Yaskawa INFORM job: DEMO_ROOF_SIDE_0625_3PAINT_23.JBI

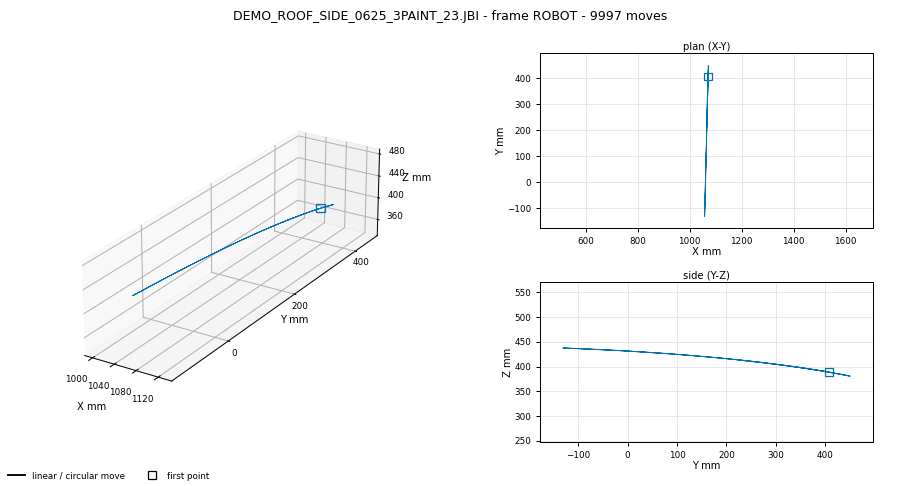
[picture p0: tool path of DEMO_ROOF_SIDE_0625_3PAINT_23.JBI in frame ROBOT, 9997 of 9997 moves have a stored position in this frame; points joined in program order, loops and branches not executed]
/JOB
//NAME DEMO_ROOF_SIDE_0625_3PAINT23
//POS
///NPOS 9997,0,0,0,0,0
///TOOL 0
///USER 0
///POSTYPE ROBOT
///RECTAN
///RCONF 1,0,0,0,0,0,0,0,0,0,0,0,0,0,0,0,0,0,0,0,0,0,0,0
C00000=1071.321,407.513,389.475,175.844,34.112,156.275
C00001=1071.313,407.267,389.517,175.839,34.102,156.273
C00002=1071.307,407.021,389.559,175.833,34.094,156.271
C00003=1071.298,406.775,389.602,175.828,34.084,156.268
C00004=1071.291,406.528,389.645,175.822,34.075,156.266
C00005=1071.284,406.282,389.687,175.818,34.066,156.264
C00006=1071.277,406.036,389.729,175.812,34.057,156.262
C00007=1071.269,405.789,389.771,175.807,34.048,156.260
C00008=1071.262,405.543,389.813,175.801,34.039,156.258
C00009=1071.254,405.297,389.855,175.796,34.030,156.256
C00010=1071.248,405.050,389.898,175.791,34.021,156.254
C00011=1071.240,404.804,389.940,175.785,34.012,156.252
C00012=1071.233,404.558,389.982,175.780,34.003,156.250
C00013=1071.225,404.311,390.025,175.775,33.995,156.248
C00014=1071.218,404.065,390.066,175.770,33.986,156.246
C00015=1071.211,403.818,390.108,175.765,33.977,156.244
C00016=1071.203,403.573,390.150,175.759,33.968,156.242
C00017=1071.196,403.326,390.192,175.754,33.959,156.240
C00018=1071.189,403.080,390.234,175.749,33.951,156.238
C00019=1071.182,402.833,390.275,175.744,33.942,156.236
C00020=1071.174,402.587,390.317,175.739,33.933,156.234
C00021=1071.166,402.341,390.359,175.733,33.925,156.232
C00022=1071.159,402.094,390.401,175.728,33.916,156.230
C00023=1071.152,401.847,390.443,175.723,33.907,156.228
C00024=1071.144,401.601,390.485,175.718,33.899,156.226
C00025=1071.137,401.354,390.526,175.713,33.890,156.224
C00026=1071.130,401.108,390.568,175.707,33.882,156.222
C00027=1071.122,400.862,390.609,175.703,33.873,156.220
C00028=1071.115,400.615,390.650,175.698,33.865,156.219
C00029=1071.109,400.370,390.692,175.692,33.856,156.217
C00030=1071.101,400.123,390.734,175.687,33.848,156.215
C00031=1071.094,399.856,390.778,175.682,33.838,156.213
C00032=1071.086,399.589,390.823,175.676,33.829,156.211
C00033=1071.078,399.323,390.868,175.671,33.820,156.208
C00034=1071.070,399.056,390.913,175.665,33.811,156.206
C00035=1071.063,398.809,390.954,175.660,33.803,156.205
C00036=1071.055,398.563,390.996,175.656,33.794,156.203
C00037=1071.049,398.316,391.038,175.650,33.786,156.201
C00038=1071.041,398.070,391.079,175.645,33.778,156.199
C00039=1071.033,397.823,391.119,175.641,33.770,156.197
C00040=1071.027,397.578,391.160,175.636,33.761,156.195
C00041=1071.019,397.331,391.201,175.630,33.753,156.193
C00042=1071.012,397.084,391.243,175.626,33.745,156.192
C00043=1071.005,396.838,391.284,175.621,33.737,156.190
C00044=1070.998,396.591,391.324,175.616,33.729,156.188
C00045=1070.991,396.345,391.365,175.611,33.720,156.186
C00046=1070.984,396.098,391.407,175.606,33.712,156.184
C00047=1070.976,395.851,391.448,175.601,33.704,156.183
C00048=1070.970,395.606,391.489,175.596,33.696,156.181
C00049=1070.962,395.359,391.530,175.591,33.688,156.179
C00050=1070.955,395.112,391.570,175.587,33.680,156.177
C00051=1070.948,394.866,391.611,175.581,33.672,156.175
C00052=1070.941,394.620,391.652,175.577,33.664,156.174
C00053=1070.934,394.372,391.692,175.572,33.656,156.172
C00054=1070.927,394.127,391.733,175.568,33.648,156.170
C00055=1070.920,393.880,391.774,175.562,33.640,156.168
C00056=1070.912,393.633,391.814,175.557,33.632,156.167
C00057=1070.905,393.387,391.855,175.553,33.624,156.165
C00058=1070.898,393.140,391.896,175.548,33.617,156.163
C00059=1070.892,392.894,391.937,175.543,33.608,156.161
C00060=1070.884,392.647,391.977,175.538,33.600,156.160
C00061=1070.877,392.401,392.018,175.534,33.593,156.158
C00062=1070.870,392.154,392.058,175.529,33.585,156.156
C00063=1070.862,391.908,392.099,175.524,33.578,156.154
C00064=1070.856,391.661,392.139,175.519,33.570,156.153
C00065=1070.849,391.414,392.179,175.515,33.562,156.151
C00066=1070.841,391.168,392.219,175.510,33.554,156.149
C00067=1070.835,390.922,392.260,175.506,33.546,156.148
C00068=1070.828,390.675,392.300,175.500,33.539,156.146
C00069=1070.820,390.428,392.340,175.496,33.531,156.144
C00070=1070.814,390.182,392.381,175.491,33.523,156.143
C00071=1070.806,389.935,392.421,175.487,33.516,156.141
C00072=1070.799,389.689,392.460,175.481,33.508,156.139
C00073=1070.793,389.442,392.501,175.477,33.501,156.138
C00074=1070.785,389.195,392.540,175.472,33.493,156.136
C00075=1070.778,388.949,392.581,175.468,33.486,156.134
C00076=1070.771,388.702,392.621,175.463,33.478,156.133
C00077=1070.764,388.455,392.661,175.459,33.471,156.131
C00078=1070.757,388.209,392.701,175.453,33.463,156.129
C00079=1070.749,387.962,392.740,175.449,33.456,156.128
C00080=1070.743,387.716,392.780,175.444,33.448,156.126
C00081=1070.735,387.469,392.820,175.440,33.441,156.124
C00082=1070.729,387.222,392.860,175.435,33.433,156.123
C00083=1070.722,386.976,392.900,175.430,33.426,156.121
C00084=1070.714,386.729,392.940,175.426,33.419,156.120
C00085=1070.708,386.483,392.980,175.421,33.411,156.118
C00086=1070.701,386.237,393.020,175.417,33.404,156.117
C00087=1070.694,385.985,393.060,175.412,33.396,156.115
C00088=1070.686,385.734,393.100,175.408,33.389,156.113
C00089=1070.680,385.483,393.141,175.402,33.382,156.112
C00090=1070.673,385.232,393.181,175.398,33.374,156.110
C00091=1070.666,384.985,393.220,175.394,33.367,156.108
C00092=1070.658,384.738,393.260,175.389,33.360,156.107
C00093=1070.652,384.492,393.300,175.385,33.352,156.105
C00094=1070.645,384.245,393.339,175.381,33.345,156.104
C00095=1070.638,383.999,393.379,175.376,33.338,156.102
C00096=1070.632,383.752,393.418,175.371,33.331,156.101
C00097=1070.625,383.505,393.458,175.366,33.323,156.099
C00098=1070.617,383.258,393.498,175.362,33.316,156.097
C00099=1070.611,383.011,393.537,175.358,33.309,156.096
C00100=1070.604,382.765,393.577,175.354,33.302,156.094
C00101=1070.597,382.518,393.615,175.349,33.295,156.093
C00102=1070.590,382.271,393.654,175.345,33.288,156.091
C00103=1070.584,382.025,393.694,175.340,33.281,156.090
C00104=1070.577,381.778,393.733,175.335,33.274,156.088
C00105=1070.570,381.532,393.773,175.331,33.266,156.087
C00106=1070.563,381.285,393.812,175.327,33.260,156.085
C00107=1070.556,381.038,393.851,175.322,33.252,156.084
C00108=1070.549,380.791,393.890,175.318,33.245,156.082
C00109=1070.543,380.544,393.930,175.314,33.239,156.081
C00110=1070.536,380.297,393.969,175.310,33.232,156.079
C00111=1070.529,380.051,394.008,175.305,33.225,156.078
C00112=1070.522,379.804,394.046,175.301,33.217,156.076
C00113=1070.515,379.557,394.085,175.296,33.211,156.075
C00114=1070.509,379.310,394.124,175.291,33.204,156.073
C00115=1070.502,379.063,394.163,175.287,33.197,156.072
C00116=1070.495,378.816,394.202,175.283,33.190,156.070
C00117=1070.488,378.570,394.241,175.279,33.183,156.069
C00118=1070.480,378.324,394.280,175.274,33.176,156.068
C00119=1070.474,378.076,394.318,175.270,33.170,156.066
C00120=1070.467,377.830,394.356,175.266,33.163,156.065
C00121=1070.460,377.583,394.395,175.262,33.156,156.063
C00122=1070.453,377.336,394.434,175.258,33.149,156.062
C00123=1070.447,377.089,394.473,175.253,33.143,156.060
C00124=1070.440,376.842,394.512,175.248,33.136,156.059
C00125=1070.433,376.595,394.551,175.244,33.129,156.057
C00126=1070.426,376.349,394.590,175.240,33.122,156.056
C00127=1070.419,376.102,394.628,175.235,33.115,156.055
C00128=1070.413,375.854,394.666,175.231,33.109,156.053
C00129=1070.406,375.607,394.705,175.227,33.102,156.052
C00130=1070.400,375.361,394.744,175.223,33.096,156.050
C00131=1070.393,375.115,394.783,175.219,33.089,156.049
C00132=1070.386,374.867,394.821,175.215,33.082,156.048
C00133=1070.380,374.620,394.860,175.210,33.075,156.046
C00134=1070.372,374.374,394.898,175.206,33.069,156.045
C00135=1070.366,374.126,394.936,175.202,33.062,156.043
C00136=1070.359,373.880,394.974,175.198,33.055,156.042
C00137=1070.353,373.633,395.013,175.194,33.049,156.041
C00138=1070.346,373.386,395.051,175.190,33.042,156.039
C00139=1070.340,373.152,395.088,175.186,33.037,156.038
C00140=1070.334,372.918,395.124,175.181,33.030,156.037
C00141=1070.327,372.684,395.160,175.177,33.024,156.035
C00142=1070.320,372.449,395.196,175.173,33.018,156.034
C00143=1070.314,372.215,395.233,175.169,33.012,156.033
C00144=1070.308,371.982,395.268,175.165,33.006,156.031
C00145=1070.301,371.747,395.305,175.161,33.000,156.030
C00146=1070.294,371.513,395.341,175.157,32.993,156.029
C00147=1070.288,371.267,395.379,175.153,32.987,156.027
C00148=1070.282,371.019,395.417,175.149,32.981,156.026
C00149=1070.274,370.773,395.455,175.145,32.974,156.025
C00150=1070.268,370.525,395.493,175.141,32.968,156.024
C00151=1070.261,370.279,395.530,175.137,32.962,156.022
C00152=1070.254,370.031,395.568,175.133,32.955,156.021
C00153=1070.248,369.785,395.607,175.129,32.949,156.019
C00154=1070.240,369.537,395.645,175.125,32.942,156.018
C00155=1070.235,369.291,395.682,175.120,32.936,156.017
C00156=1070.227,369.043,395.720,175.116,32.930,156.016
C00157=1070.221,368.796,395.758,175.112,32.924,156.014
C00158=1070.214,368.550,395.795,175.108,32.917,156.013
C00159=1070.208,368.302,395.833,175.104,32.911,156.012
C00160=1070.201,368.055,395.872,175.100,32.905,156.010
C00161=1070.194,367.809,395.909,175.096,32.898,156.009
C00162=1070.188,367.561,395.947,175.092,32.892,156.008
C00163=1070.181,367.315,395.985,175.088,32.886,156.006
C00164=1070.175,367.068,396.023,175.084,32.880,156.005
C00165=1070.168,366.821,396.059,175.080,32.874,156.004
C00166=1070.162,366.573,396.097,175.076,32.867,156.003
C00167=1070.154,366.326,396.135,175.072,32.861,156.001
C00168=1070.149,366.079,396.173,175.068,32.855,156.000
C00169=1070.141,365.832,396.210,175.064,32.849,155.999
C00170=1070.135,365.585,396.248,175.060,32.842,155.997
C00171=1070.128,365.338,396.285,175.056,32.837,155.996
C00172=1070.122,365.091,396.323,175.052,32.830,155.995
C00173=1070.115,364.844,396.360,175.048,32.824,155.994
C00174=1070.109,364.597,396.398,175.044,32.818,155.992
C00175=1070.102,364.350,396.435,175.040,32.812,155.991
C00176=1070.096,364.103,396.472,175.036,32.806,155.990
C00177=1070.089,363.855,396.510,175.032,32.800,155.989
C00178=1070.083,363.609,396.547,175.028,32.794,155.987
C00179=1070.076,363.361,396.584,175.024,32.788,155.986
C00180=1070.069,363.115,396.621,175.020,32.782,155.985
C00181=1070.063,362.867,396.659,175.016,32.776,155.984
C00182=1070.056,362.620,396.695,175.012,32.770,155.982
C00183=1070.049,362.373,396.733,175.008,32.764,155.981
C00184=1070.043,362.126,396.769,175.004,32.758,155.980
C00185=1070.036,361.879,396.808,175.000,32.752,155.979
C00186=1070.030,361.632,396.844,174.996,32.746,155.978
C00187=1070.023,361.384,396.882,174.992,32.740,155.976
C00188=1070.016,361.137,396.918,174.988,32.734,155.975
C00189=1070.010,360.890,396.954,174.984,32.728,155.974
C00190=1070.003,360.643,396.993,174.980,32.722,155.973
C00191=1069.997,360.396,397.029,174.976,32.716,155.971
C00192=1069.990,360.149,397.067,174.972,32.710,155.970
C00193=1069.983,359.902,397.103,174.969,32.705,155.969
C00194=1069.977,359.655,397.139,174.965,32.699,155.968
C00195=1069.971,359.429,397.174,174.961,32.694,155.967
C00196=1069.965,359.203,397.207,174.958,32.688,155.966
C00197=1069.960,358.978,397.240,174.955,32.683,155.965
C00198=1069.953,358.753,397.274,174.951,32.677,155.963
C00199=1069.947,358.527,397.308,174.948,32.672,155.962
C00200=1069.941,358.301,397.341,174.944,32.667,155.961
C00201=1069.936,358.075,397.375,174.941,32.661,155.960
C00202=1069.929,357.850,397.408,174.937,32.656,155.959
C00203=1069.922,357.603,397.445,174.933,32.651,155.958
C00204=1069.916,357.356,397.481,174.929,32.645,155.957
C00205=1069.909,357.108,397.518,174.925,32.639,155.956
C00206=1069.903,356.861,397.555,174.922,32.633,155.955
C00207=1069.896,356.614,397.591,174.918,32.628,155.953
C00208=1069.890,356.367,397.627,174.914,32.622,155.952
C00209=1069.883,356.119,397.664,174.910,32.616,155.951
C00210=1069.877,355.872,397.701,174.906,32.610,155.950
C00211=1069.871,355.625,397.737,174.902,32.605,155.949
C00212=1069.864,355.378,397.774,174.898,32.599,155.948
C00213=1069.857,355.130,397.810,174.895,32.594,155.946
C00214=1069.851,354.883,397.847,174.891,32.588,155.945
C00215=1069.845,354.636,397.883,174.887,32.582,155.944
C00216=1069.839,354.389,397.919,174.883,32.576,155.943
C00217=1069.832,354.141,397.955,174.880,32.571,155.942
C00218=1069.825,353.894,397.992,174.876,32.565,155.941
C00219=1069.819,353.647,398.029,174.873,32.560,155.940
C00220=1069.813,353.400,398.065,174.869,32.554,155.939
C00221=1069.806,353.152,398.100,174.865,32.548,155.937
C00222=1069.799,352.905,398.137,174.861,32.543,155.936
C00223=1069.793,352.658,398.173,174.857,32.537,155.935
C00224=1069.786,352.410,398.210,174.853,32.532,155.934
C00225=1069.780,352.163,398.246,174.850,32.526,155.933
C00226=1069.774,351.916,398.282,174.846,32.521,155.932
C00227=1069.767,351.669,398.318,174.842,32.515,155.931
C00228=1069.761,351.421,398.354,174.838,32.509,155.930
C00229=1069.754,351.174,398.390,174.834,32.504,155.929
C00230=1069.748,350.927,398.425,174.831,32.499,155.927
C00231=1069.741,350.680,398.462,174.828,32.493,155.926
C00232=1069.735,350.431,398.498,174.824,32.488,155.925
C00233=1069.728,350.184,398.534,174.820,32.482,155.924
C00234=1069.722,349.937,398.569,174.817,32.477,155.923
C00235=1069.715,349.690,398.606,174.813,32.471,155.922
C00236=1069.709,349.442,398.642,174.809,32.466,155.921
C00237=1069.702,349.195,398.678,174.805,32.460,155.920
C00238=1069.696,348.948,398.713,174.801,32.455,155.919
C00239=1069.690,348.700,398.749,174.798,32.450,155.918
C00240=1069.683,348.453,398.785,174.794,32.444,155.916
C00241=1069.677,348.206,398.821,174.790,32.439,155.915
C00242=1069.671,347.959,398.857,174.787,32.433,155.914
C00243=1069.664,347.711,398.892,174.784,32.428,155.913
C00244=1069.658,347.464,398.928,174.780,32.423,155.912
C00245=1069.651,347.216,398.963,174.776,32.417,155.911
C00246=1069.645,346.969,398.999,174.773,32.412,155.910
C00247=1069.639,346.722,399.035,174.769,32.407,155.909
C00248=1069.632,346.474,399.070,174.765,32.401,155.908
C00249=1069.626,346.226,399.106,174.761,32.396,155.907
C00250=1069.619,345.979,399.141,174.758,32.391,155.906
C00251=1069.614,345.756,399.174,174.754,32.386,155.905
C00252=1069.607,345.532,399.206,174.751,32.381,155.904
C00253=1069.602,345.309,399.238,174.749,32.376,155.903
C00254=1069.596,345.085,399.270,174.745,32.371,155.902
C00255=1069.591,344.861,399.302,174.742,32.366,155.901
C00256=1069.585,344.638,399.334,174.739,32.362,155.900
C00257=1069.579,344.413,399.367,174.735,32.357,155.899
C00258=1069.574,344.190,399.398,174.732,32.352,155.898
C00259=1069.567,343.942,399.433,174.728,32.347,155.897
C00260=1069.561,343.695,399.469,174.725,32.341,155.896
C00261=1069.554,343.447,399.504,174.721,32.337,155.895
C00262=1069.548,343.200,399.540,174.717,32.331,155.894
C00263=1069.541,342.952,399.575,174.714,32.326,155.893
C00264=1069.535,342.706,399.610,174.711,32.320,155.892
C00265=1069.528,342.458,399.645,174.707,32.316,155.891
C00266=1069.522,342.211,399.680,174.703,32.310,155.890
C00267=1069.515,341.963,399.716,174.700,32.305,155.889
C00268=1069.509,341.715,399.750,174.696,32.300,155.888
C00269=1069.503,341.468,399.786,174.692,32.295,155.887
C00270=1069.496,341.220,399.821,174.689,32.289,155.886
C00271=1069.490,340.974,399.856,174.685,32.285,155.885
C00272=1069.484,340.726,399.891,174.683,32.279,155.884
C00273=1069.478,340.478,399.926,174.679,32.274,155.883
C00274=1069.471,340.231,399.961,174.675,32.269,155.882
C00275=1069.465,339.984,399.996,174.672,32.264,155.881
C00276=1069.459,339.736,400.031,174.668,32.259,155.880
C00277=1069.452,339.488,400.066,174.664,32.254,155.879
C00278=1069.445,339.241,400.101,174.661,32.248,155.878
C00279=1069.440,338.993,400.136,174.657,32.243,155.877
C00280=1069.433,338.746,400.171,174.655,32.238,155.876
C00281=1069.427,338.499,400.206,174.651,32.233,155.875
C00282=1069.420,338.251,400.240,174.647,32.228,155.874
C00283=1069.415,338.004,400.276,174.644,32.223,155.873
C00284=1069.408,337.756,400.310,174.640,32.218,155.872
C00285=1069.402,337.508,400.345,174.637,32.213,155.871
C00286=1069.396,337.261,400.379,174.633,32.208,155.870
C00287=1069.389,337.014,400.414,174.629,32.203,155.869
C00288=1069.382,336.766,400.449,174.627,32.198,155.868
C00289=1069.376,336.518,400.484,174.623,32.193,155.867
C00290=1069.370,336.271,400.518,174.620,32.188,155.866
C00291=1069.363,336.023,400.552,174.616,32.183,155.865
C00292=1069.357,335.776,400.588,174.612,32.178,155.864
C00293=1069.351,335.528,400.622,174.609,32.173,155.863
C00294=1069.344,335.280,400.656,174.605,32.168,155.862
C00295=1069.338,335.033,400.692,174.602,32.163,155.861
C00296=1069.332,334.785,400.726,174.599,32.158,155.860
C00297=1069.326,334.537,400.760,174.596,32.153,155.859
C00298=1069.320,334.291,400.795,174.592,32.148,155.858
C00299=1069.313,334.043,400.829,174.588,32.143,155.858
C00300=1069.307,333.795,400.864,174.585,32.138,155.857
C00301=1069.301,333.548,400.898,174.581,32.133,155.856
C00302=1069.294,333.300,400.932,174.578,32.128,155.855
C00303=1069.288,333.053,400.967,174.575,32.123,155.854
C00304=1069.282,332.805,401.002,174.572,32.118,155.853
C00305=1069.276,332.558,401.036,174.568,32.113,155.852
C00306=1069.269,332.310,401.069,174.565,32.109,155.851
C00307=1069.263,332.083,401.101,174.562,32.104,155.850
C00308=1069.257,331.858,401.133,174.558,32.099,155.849
C00309=1069.252,331.631,401.164,174.555,32.095,155.848
C00310=1069.247,331.405,401.195,174.553,32.091,155.847
C00311=1069.241,331.179,401.226,174.550,32.086,155.847
C00312=1069.235,330.953,401.257,174.546,32.082,155.846
C00313=1069.229,330.727,401.289,174.543,32.077,155.845
C00314=1069.223,330.501,401.320,174.540,32.073,155.844
C00315=1069.216,330.253,401.354,174.537,32.068,155.843
C00316=1069.210,330.006,401.388,174.533,32.063,155.842
C00317=1069.204,329.757,401.421,174.530,32.058,155.841
C00318=1069.198,329.510,401.455,174.527,32.054,155.840
C00319=1069.191,329.262,401.490,174.523,32.049,155.840
C00320=1069.185,329.015,401.523,174.520,32.045,155.839
C00321=1069.178,328.767,401.558,174.516,32.040,155.838
C00322=1069.172,328.520,401.592,174.513,32.035,155.837
C00323=1069.164,328.234,401.630,174.509,32.029,155.836
C00324=1069.157,327.949,401.669,174.506,32.024,155.835
C00325=1069.150,327.663,401.708,174.502,32.019,155.834
C00326=1069.142,327.378,401.747,174.498,32.013,155.833
C00327=1069.136,327.130,401.782,174.494,32.008,155.832
C00328=1069.129,326.882,401.814,174.491,32.003,155.831
C00329=1069.123,326.634,401.849,174.488,31.999,155.830
C00330=1069.117,326.387,401.883,174.485,31.994,155.829
C00331=1069.111,326.139,401.916,174.482,31.989,155.828
C00332=1069.104,325.891,401.950,174.478,31.985,155.827
C00333=1069.098,325.644,401.984,174.475,31.980,155.826
C00334=1069.092,325.396,402.017,174.471,31.975,155.825
C00335=1069.085,325.149,402.051,174.468,31.971,155.824
C00336=1069.079,324.901,402.084,174.465,31.966,155.824
C00337=1069.072,324.653,402.118,174.462,31.961,155.823
C00338=1069.066,324.406,402.152,174.459,31.957,155.822
C00339=1069.061,324.158,402.185,174.455,31.952,155.821
C00340=1069.054,323.910,402.219,174.452,31.947,155.820
C00341=1069.048,323.662,402.252,174.448,31.943,155.819
C00342=1069.041,323.415,402.286,174.446,31.938,155.818
C00343=1069.035,323.167,402.320,174.442,31.933,155.817
C00344=1069.029,322.920,402.353,174.439,31.929,155.817
C00345=1069.023,322.672,402.386,174.436,31.924,155.816
C00346=1069.016,322.424,402.420,174.432,31.919,155.815
C00347=1069.010,322.176,402.454,174.429,31.915,155.814
C00348=1069.004,321.929,402.486,174.426,31.910,155.813
C00349=1068.998,321.681,402.520,174.423,31.905,155.812
C00350=1068.991,321.433,402.553,174.420,31.901,155.811
C00351=1068.986,321.185,402.587,174.416,31.896,155.810
C00352=1068.979,320.938,402.620,174.413,31.891,155.809
C00353=1068.974,320.690,402.654,174.410,31.887,155.809
C00354=1068.967,320.443,402.686,174.407,31.882,155.808
C00355=1068.961,320.194,402.720,174.404,31.878,155.807
C00356=1068.955,319.947,402.754,174.400,31.873,155.806
C00357=1068.948,319.700,402.786,174.397,31.868,155.805
C00358=1068.943,319.452,402.820,174.394,31.864,155.804
C00359=1068.936,319.204,402.852,174.391,31.859,155.803
C00360=1068.931,318.957,402.886,174.388,31.855,155.803
C00361=1068.924,318.708,402.920,174.385,31.850,155.802
C00362=1068.918,318.461,402.953,174.381,31.845,155.801
C00363=1068.913,318.251,402.981,174.378,31.841,155.800
C00364=1068.907,318.041,403.009,174.376,31.838,155.799
C00365=1068.903,317.830,403.037,174.374,31.833,155.799
C00366=1068.898,317.620,403.065,174.371,31.830,155.798
C00367=1068.892,317.410,403.093,174.368,31.825,155.797
C00368=1068.888,317.199,403.121,174.365,31.822,155.796
C00369=1068.882,316.989,403.149,174.362,31.817,155.796
C00370=1068.877,316.779,403.177,174.360,31.814,155.795
C00371=1068.871,316.531,403.210,174.357,31.809,155.794
C00372=1068.865,316.283,403.243,174.354,31.805,155.793
C00373=1068.859,316.036,403.276,174.351,31.800,155.792
C00374=1068.853,315.788,403.309,174.347,31.795,155.791
C00375=1068.847,315.540,403.342,174.344,31.791,155.791
C00376=1068.841,315.293,403.375,174.341,31.786,155.790
C00377=1068.835,315.045,403.408,174.338,31.781,155.789
C00378=1068.829,314.797,403.441,174.335,31.777,155.788
C00379=1068.823,314.549,403.474,174.332,31.772,155.787
C00380=1068.817,314.302,403.507,174.329,31.768,155.786
C00381=1068.811,314.053,403.539,174.325,31.764,155.785
C00382=1068.804,313.805,403.572,174.323,31.759,155.785
C00383=1068.798,313.558,403.605,174.320,31.755,155.784
C00384=1068.791,313.310,403.638,174.316,31.750,155.783
C00385=1068.785,313.062,403.670,174.313,31.746,155.782
C00386=1068.779,312.814,403.702,174.310,31.742,155.781
C00387=1068.773,312.567,403.735,174.307,31.737,155.781
C00388=1068.766,312.319,403.767,174.304,31.733,155.780
C00389=1068.760,312.071,403.799,174.301,31.728,155.779
C00390=1068.754,311.823,403.832,174.297,31.724,155.778
C00391=1068.747,311.576,403.865,174.294,31.719,155.777
C00392=1068.741,311.328,403.897,174.291,31.715,155.776
C00393=1068.735,311.080,403.930,174.289,31.711,155.776
C00394=1068.729,310.833,403.962,174.285,31.706,155.775
C00395=1068.723,310.584,403.994,174.282,31.702,155.774
C00396=1068.716,310.337,404.027,174.279,31.697,155.773
C00397=1068.709,310.089,404.059,174.275,31.693,155.772
C00398=1068.703,309.841,404.091,174.273,31.689,155.772
C00399=1068.697,309.594,404.124,174.270,31.684,155.771
C00400=1068.691,309.345,404.156,174.267,31.680,155.770
C00401=1068.685,309.098,404.189,174.263,31.676,155.769
C00402=1068.679,308.850,404.221,174.260,31.671,155.768
C00403=1068.672,308.602,404.253,174.258,31.667,155.768
C00404=1068.666,308.354,404.285,174.255,31.663,155.767
C00405=1068.660,308.107,404.318,174.251,31.658,155.766
C00406=1068.654,307.859,404.349,174.248,31.654,155.765
C00407=1068.648,307.611,404.382,174.245,31.649,155.764
C00408=1068.642,307.363,404.414,174.243,31.645,155.764
C00409=1068.635,307.115,404.446,174.239,31.641,155.763
C00410=1068.629,306.868,404.478,174.236,31.636,155.762
C00411=1068.623,306.619,404.510,174.233,31.632,155.761
C00412=1068.617,306.372,404.543,174.230,31.628,155.760
C00413=1068.611,306.124,404.575,174.227,31.623,155.760
C00414=1068.604,305.876,404.606,174.224,31.619,155.759
C00415=1068.598,305.629,404.639,174.221,31.615,155.758
C00416=1068.592,305.381,404.671,174.218,31.610,155.757
C00417=1068.586,305.132,404.703,174.215,31.606,155.756
C00418=1068.580,304.885,404.734,174.212,31.602,155.756
C00419=1068.575,304.658,404.764,174.209,31.597,155.755
C00420=1068.569,304.430,404.793,174.206,31.594,155.754
C00421=1068.564,304.203,404.823,174.203,31.589,155.753
C00422=1068.558,303.975,404.852,174.201,31.586,155.753
C00423=1068.552,303.748,404.881,174.199,31.581,155.752
C00424=1068.547,303.521,404.910,174.196,31.578,155.751
C00425=1068.541,303.293,404.940,174.193,31.573,155.750
C00426=1068.535,303.066,404.969,174.190,31.570,155.750
C00427=1068.529,302.817,405.001,174.187,31.565,155.749
C00428=1068.523,302.569,405.033,174.184,31.561,155.748
C00429=1068.518,302.322,405.065,174.181,31.557,155.747
C00430=1068.511,302.074,405.096,174.178,31.552,155.747
C00431=1068.505,301.826,405.129,174.175,31.548,155.746
C00432=1068.499,301.579,405.160,174.173,31.544,155.745
C00433=1068.493,301.331,405.192,174.169,31.539,155.744
C00434=1068.487,301.083,405.224,174.166,31.535,155.743
C00435=1068.481,300.835,405.256,174.163,31.531,155.743
C00436=1068.475,300.587,405.288,174.160,31.526,155.742
C00437=1068.469,300.339,405.319,174.158,31.522,155.741
C00438=1068.463,300.092,405.351,174.155,31.518,155.740
C00439=1068.457,299.843,405.383,174.152,31.514,155.739
C00440=1068.451,299.596,405.414,174.148,31.509,155.739
C00441=1068.445,299.348,405.446,174.146,31.505,155.738
C00442=1068.440,299.099,405.477,174.143,31.500,155.737
C00443=1068.433,298.852,405.508,174.140,31.496,155.736
C00444=1068.427,298.604,405.540,174.137,31.492,155.735
C00445=1068.422,298.356,405.572,174.134,31.488,155.735
C00446=1068.415,298.108,405.603,174.132,31.483,155.734
C00447=1068.410,297.861,405.635,174.128,31.479,155.733
C00448=1068.404,297.612,405.667,174.125,31.474,155.732
C00449=1068.397,297.364,405.698,174.122,31.470,155.731
C00450=1068.392,297.116,405.729,174.120,31.466,155.731
C00451=1068.385,296.869,405.761,174.117,31.462,155.730
C00452=1068.380,296.621,405.792,174.114,31.457,155.729
C00453=1068.374,296.373,405.823,174.111,31.453,155.728
C00454=1068.368,296.124,405.855,174.108,31.449,155.728
C00455=1068.361,295.877,405.886,174.105,31.445,155.727
C00456=1068.355,295.629,405.917,174.102,31.440,155.726
C00457=1068.350,295.381,405.949,174.099,31.436,155.725
C00458=1068.343,295.133,405.980,174.096,31.432,155.725
C00459=1068.337,294.885,406.010,174.094,31.428,155.724
C00460=1068.331,294.637,406.042,174.091,31.424,155.723
C00461=1068.325,294.389,406.073,174.088,31.419,155.722
C00462=1068.319,294.141,406.104,174.085,31.416,155.722
C00463=1068.313,293.893,406.136,174.082,31.411,155.721
C00464=1068.307,293.645,406.167,174.079,31.407,155.720
C00465=1068.300,293.397,406.198,174.076,31.402,155.719
C00466=1068.294,293.150,406.228,174.073,31.399,155.719
C00467=1068.288,292.901,406.260,174.070,31.394,155.718
C00468=1068.282,292.654,406.291,174.068,31.390,155.717
C00469=1068.276,292.406,406.322,174.065,31.386,155.716
C00470=1068.270,292.158,406.353,174.062,31.382,155.716
C00471=1068.264,291.910,406.385,174.059,31.378,155.715
C00472=1068.258,291.662,406.415,174.057,31.373,155.714
C00473=1068.252,291.413,406.446,174.054,31.370,155.713
C00474=1068.246,291.166,406.477,174.051,31.365,155.712
C00475=1068.240,290.946,406.504,174.048,31.361,155.712
C00476=1068.235,290.726,406.532,174.045,31.358,155.711
C00477=1068.230,290.505,406.559,174.044,31.354,155.710
C00478=1068.225,290.285,406.586,174.041,31.350,155.710
C00479=1068.219,290.066,406.614,174.038,31.346,155.709
C00480=1068.214,289.846,406.641,174.035,31.343,155.708
C00481=1068.208,289.626,406.668,174.034,31.339,155.708
C00482=1068.203,289.405,406.696,174.031,31.336,155.707
C00483=1068.197,289.158,406.726,174.028,31.332,155.706
C00484=1068.191,288.910,406.758,174.025,31.327,155.706
C00485=1068.185,288.662,406.788,174.022,31.323,155.705
C00486=1068.178,288.413,406.819,174.020,31.319,155.704
C00487=1068.173,288.165,406.849,174.017,31.315,155.703
C00488=1068.166,287.917,406.880,174.014,31.311,155.703
C00489=1068.160,287.670,406.911,174.011,31.307,155.702
C00490=1068.154,287.422,406.941,174.009,31.303,155.701
C00491=1068.148,287.173,406.972,174.006,31.299,155.700
C00492=1068.142,286.926,407.002,174.003,31.294,155.700
C00493=1068.136,286.677,407.033,174.000,31.290,155.699
C00494=1068.130,286.429,407.063,173.997,31.286,155.698
C00495=1068.124,286.181,407.094,173.994,31.282,155.698
C00496=1068.117,285.933,407.124,173.991,31.278,155.697
C00497=1068.112,285.685,407.155,173.988,31.274,155.696
C00498=1068.106,285.437,407.185,173.986,31.270,155.695
C00499=1068.099,285.189,407.216,173.983,31.265,155.695
C00500=1068.094,284.941,407.246,173.980,31.262,155.694
C00501=1068.088,284.693,407.277,173.977,31.257,155.693
C00502=1068.081,284.445,407.307,173.975,31.253,155.692
C00503=1068.076,284.197,407.338,173.972,31.249,155.692
C00504=1068.069,283.949,407.367,173.969,31.245,155.691
C00505=1068.063,283.701,407.398,173.966,31.241,155.690
C00506=1068.057,283.453,407.428,173.964,31.237,155.689
C00507=1068.051,283.205,407.459,173.961,31.233,155.689
C00508=1068.045,282.957,407.490,173.958,31.228,155.688
C00509=1068.039,282.709,407.520,173.955,31.225,155.687
C00510=1068.033,282.461,407.550,173.953,31.220,155.686
C00511=1068.027,282.212,407.580,173.950,31.216,155.686
C00512=1068.021,281.964,407.611,173.948,31.212,155.685
C00513=1068.015,281.716,407.641,173.945,31.208,155.684
C00514=1068.009,281.468,407.671,173.943,31.204,155.684
C00515=1068.003,281.221,407.701,173.940,31.200,155.683
C00516=1067.997,280.972,407.731,173.937,31.196,155.682
C00517=1067.991,280.724,407.761,173.934,31.192,155.681
C00518=1067.985,280.476,407.792,173.932,31.187,155.681
C00519=1067.979,280.228,407.822,173.929,31.184,155.680
C00520=1067.974,279.980,407.852,173.926,31.180,155.679
C00521=1067.967,279.732,407.882,173.923,31.175,155.678
C00522=1067.961,279.484,407.912,173.921,31.172,155.678
C00523=1067.955,279.235,407.942,173.918,31.167,155.677
C00524=1067.949,278.988,407.972,173.915,31.163,155.676
C00525=1067.942,278.739,408.002,173.912,31.159,155.676
C00526=1067.937,278.491,408.032,173.910,31.155,155.675
C00527=1067.930,278.243,408.062,173.907,31.151,155.674
C00528=1067.925,277.995,408.091,173.904,31.147,155.673
C00529=1067.919,277.747,408.122,173.901,31.143,155.673
C00530=1067.913,277.499,408.152,173.899,31.139,155.672
C00531=1067.907,277.284,408.178,173.897,31.135,155.671
C00532=1067.902,277.069,408.203,173.894,31.132,155.671
C00533=1067.897,276.854,408.229,173.892,31.128,155.670
C00534=1067.891,276.639,408.255,173.890,31.125,155.669
C00535=1067.886,276.425,408.281,173.888,31.121,155.669
C00536=1067.881,276.209,408.307,173.885,31.118,155.668
C00537=1067.876,275.995,408.332,173.883,31.115,155.668
C00538=1067.870,275.780,408.358,173.880,31.111,155.667
C00539=1067.865,275.531,408.388,173.878,31.107,155.666
C00540=1067.859,275.284,408.418,173.875,31.103,155.666
C00541=1067.853,275.036,408.447,173.872,31.099,155.665
C00542=1067.847,274.787,408.477,173.870,31.094,155.664
C00543=1067.841,274.540,408.507,173.867,31.091,155.663
C00544=1067.835,274.291,408.537,173.865,31.086,155.663
C00545=1067.829,274.043,408.566,173.862,31.083,155.662
C00546=1067.822,273.794,408.596,173.860,31.078,155.661
C00547=1067.817,273.546,408.626,173.857,31.074,155.660
C00548=1067.811,273.298,408.655,173.854,31.071,155.660
C00549=1067.805,273.050,408.685,173.851,31.066,155.659
C00550=1067.799,272.802,408.714,173.849,31.062,155.658
C00551=1067.793,272.554,408.744,173.846,31.058,155.658
C00552=1067.787,272.305,408.773,173.843,31.054,155.657
C00553=1067.780,272.058,408.803,173.840,31.050,155.656
C00554=1067.775,271.809,408.832,173.839,31.046,155.655
C00555=1067.769,271.561,408.861,173.836,31.042,155.655
C00556=1067.763,271.313,408.891,173.833,31.038,155.654
C00557=1067.756,271.065,408.921,173.831,31.034,155.653
C00558=1067.751,270.817,408.950,173.828,31.030,155.653
C00559=1067.745,270.569,408.979,173.825,31.026,155.652
C00560=1067.738,270.321,409.009,173.822,31.022,155.651
C00561=1067.733,270.072,409.038,173.820,31.018,155.650
C00562=1067.727,269.824,409.067,173.818,31.014,155.650
C00563=1067.721,269.576,409.097,173.815,31.010,155.649
C00564=1067.715,269.327,409.126,173.812,31.006,155.648
C00565=1067.709,269.079,409.155,173.810,31.002,155.648
C00566=1067.703,268.831,409.185,173.807,30.998,155.647
C00567=1067.697,268.583,409.214,173.804,30.994,155.646
C00568=1067.691,268.335,409.243,173.802,30.990,155.646
C00569=1067.684,268.087,409.272,173.800,30.986,155.645
C00570=1067.679,267.838,409.301,173.797,30.982,155.644
C00571=1067.673,267.590,409.330,173.794,30.978,155.644
C00572=1067.666,267.342,409.359,173.792,30.974,155.643
C00573=1067.660,267.094,409.388,173.789,30.970,155.642
C00574=1067.655,266.845,409.418,173.786,30.966,155.641
C00575=1067.648,266.597,409.447,173.783,30.962,155.641
C00576=1067.642,266.349,409.476,173.782,30.958,155.640
C00577=1067.636,266.101,409.505,173.779,30.954,155.639
C00578=1067.630,265.852,409.535,173.776,30.950,155.639
C00579=1067.624,265.604,409.564,173.774,30.946,155.638
C00580=1067.618,265.356,409.593,173.771,30.942,155.637
C00581=1067.612,265.107,409.621,173.769,30.938,155.636
C00582=1067.606,264.859,409.651,173.766,30.934,155.636
C00583=1067.600,264.611,409.680,173.764,30.930,155.635
C00584=1067.594,264.363,409.709,173.761,30.926,155.634
C00585=1067.588,264.115,409.738,173.758,30.922,155.634
C00586=1067.582,263.867,409.766,173.756,30.918,155.633
C00587=1067.578,263.653,409.792,173.754,30.915,155.632
C00588=1067.572,263.440,409.817,173.752,30.911,155.632
C00589=1067.567,263.227,409.841,173.749,30.908,155.631
C00590=1067.561,263.014,409.866,173.748,30.904,155.631
C00591=1067.556,262.801,409.890,173.745,30.901,155.630
C00592=1067.551,262.588,409.915,173.743,30.898,155.629
C00593=1067.545,262.374,409.939,173.741,30.894,155.629
C00594=1067.540,262.162,409.964,173.739,30.891,155.628
C00595=1067.534,261.914,409.993,173.736,30.887,155.627
C00596=1067.528,261.665,410.021,173.733,30.883,155.627
C00597=1067.522,261.417,410.050,173.731,30.879,155.626
C00598=1067.516,261.168,410.079,173.729,30.875,155.625
C00599=1067.510,260.920,410.108,173.726,30.871,155.625
C00600=1067.504,260.671,410.136,173.723,30.867,155.624
C00601=1067.497,260.423,410.165,173.721,30.863,155.623
C00602=1067.491,260.175,410.194,173.719,30.860,155.623
C00603=1067.485,259.927,410.222,173.716,30.855,155.622
C00604=1067.479,259.679,410.251,173.713,30.851,155.621
C00605=1067.473,259.430,410.279,173.711,30.848,155.621
C00606=1067.467,259.182,410.308,173.709,30.844,155.620
C00607=1067.461,258.933,410.336,173.706,30.839,155.619
C00608=1067.455,258.685,410.365,173.704,30.836,155.618
C00609=1067.449,258.438,410.393,173.701,30.832,155.618
C00610=1067.443,258.189,410.421,173.698,30.828,155.617
C00611=1067.436,257.941,410.450,173.696,30.824,155.616
C00612=1067.430,257.692,410.478,173.694,30.820,155.616
C00613=1067.424,257.444,410.507,173.691,30.816,155.615
C00614=1067.419,257.196,410.535,173.688,30.812,155.614
C00615=1067.413,256.947,410.564,173.687,30.808,155.614
C00616=1067.406,256.699,410.592,173.684,30.804,155.613
C00617=1067.400,256.450,410.620,173.681,30.800,155.612
C00618=1067.394,256.202,410.649,173.678,30.796,155.612
C00619=1067.388,255.954,410.677,173.677,30.792,155.611
C00620=1067.382,255.706,410.706,173.674,30.788,155.610
C00621=1067.376,255.457,410.734,173.671,30.784,155.610
C00622=1067.370,255.210,410.762,173.669,30.780,155.609
C00623=1067.364,254.961,410.791,173.667,30.776,155.608
C00624=1067.358,254.712,410.819,173.664,30.772,155.607
C00625=1067.352,254.463,410.847,173.662,30.769,155.607
C00626=1067.347,254.216,410.876,173.659,30.764,155.606
C00627=1067.340,253.968,410.904,173.657,30.760,155.605
C00628=1067.334,253.719,410.932,173.654,30.757,155.605
C00629=1067.329,253.471,410.960,173.652,30.752,155.604
C00630=1067.323,253.222,410.988,173.650,30.749,155.603
C00631=1067.316,252.974,411.017,173.647,30.745,155.603
C00632=1067.310,252.726,411.045,173.645,30.740,155.602
C00633=1067.304,252.477,411.073,173.642,30.736,155.601
C00634=1067.298,252.229,411.101,173.640,30.733,155.600
C00635=1067.293,251.981,411.129,173.638,30.728,155.600
C00636=1067.286,251.732,411.157,173.635,30.724,155.599
C00637=1067.281,251.484,411.185,173.633,30.721,155.598
C00638=1067.275,251.235,411.213,173.631,30.716,155.598
C00639=1067.269,250.987,411.242,173.628,30.712,155.597
C00640=1067.263,250.739,411.269,173.625,30.709,155.596
C00641=1067.257,250.490,411.297,173.624,30.704,155.596
C00642=1067.252,250.242,411.325,173.621,30.700,155.595
C00643=1067.246,250.028,411.350,173.619,30.697,155.594
C00644=1067.241,249.814,411.373,173.616,30.693,155.594
C00645=1067.236,249.599,411.399,173.615,30.690,155.593
C00646=1067.231,249.385,411.422,173.613,30.687,155.592
C00647=1067.226,249.171,411.446,173.611,30.683,155.592
C00648=1067.221,248.956,411.471,173.608,30.680,155.591
C00649=1067.216,248.742,411.495,173.607,30.676,155.591
C00650=1067.211,248.527,411.519,173.605,30.673,155.590
C00651=1067.205,248.279,411.546,173.602,30.669,155.589
C00652=1067.199,248.031,411.574,173.600,30.665,155.589
C00653=1067.193,247.783,411.602,173.598,30.661,155.588
C00654=1067.187,247.534,411.630,173.595,30.656,155.587
C00655=1067.182,247.286,411.658,173.593,30.653,155.586
C00656=1067.175,247.038,411.686,173.591,30.649,155.586
C00657=1067.170,246.789,411.714,173.588,30.644,155.585
C00658=1067.164,246.540,411.742,173.586,30.641,155.584
C00659=1067.158,246.292,411.769,173.584,30.636,155.584
C00660=1067.152,246.044,411.797,173.581,30.632,155.583
C00661=1067.146,245.796,411.825,173.578,30.629,155.582
C00662=1067.140,245.547,411.853,173.577,30.625,155.582
C00663=1067.135,245.299,411.880,173.574,30.620,155.581
C00664=1067.129,245.050,411.908,173.571,30.616,155.580
C00665=1067.123,244.802,411.935,173.570,30.613,155.580
C00666=1067.117,244.553,411.963,173.567,30.608,155.579
C00667=1067.111,244.305,411.990,173.564,30.604,155.578
C00668=1067.104,244.057,412.018,173.563,30.601,155.577
C00669=1067.099,243.809,412.046,173.560,30.596,155.577
C00670=1067.092,243.560,412.073,173.557,30.592,155.576
C00671=1067.087,243.312,412.101,173.556,30.589,155.575
C00672=1067.081,243.062,412.128,173.553,30.584,155.575
C00673=1067.075,242.814,412.156,173.551,30.581,155.574
C00674=1067.069,242.567,412.183,173.549,30.577,155.573
C00675=1067.064,242.317,412.211,173.546,30.572,155.572
C00676=1067.058,242.070,412.238,173.544,30.569,155.572
C00677=1067.051,241.821,412.265,173.542,30.565,155.571
C00678=1067.045,241.573,412.293,173.539,30.561,155.571
C00679=1067.039,241.323,412.320,173.537,30.557,155.570
C00680=1067.033,241.076,412.348,173.535,30.553,155.569
C00681=1067.027,240.827,412.375,173.533,30.549,155.568
C00682=1067.021,240.579,412.402,173.530,30.545,155.568
C00683=1067.015,240.330,412.430,173.528,30.541,155.567
C00684=1067.009,240.082,412.457,173.526,30.537,155.566
C00685=1067.003,239.833,412.484,173.523,30.533,155.566
C00686=1066.997,239.585,412.511,173.521,30.529,155.565
C00687=1066.992,239.336,412.539,173.519,30.525,155.564
C00688=1066.985,239.088,412.566,173.516,30.521,155.564
C00689=1066.979,238.839,412.593,173.515,30.517,155.563
C00690=1066.973,238.590,412.620,173.512,30.513,155.562
C00691=1066.967,238.343,412.647,173.509,30.509,155.561
C00692=1066.962,238.094,412.675,173.508,30.505,155.561
C00693=1066.955,237.845,412.702,173.505,30.501,155.560
C00694=1066.949,237.597,412.729,173.503,30.497,155.559
C00695=1066.943,237.348,412.756,173.501,30.493,155.559
C00696=1066.937,237.100,412.783,173.498,30.489,155.558
C00697=1066.931,236.852,412.810,173.496,30.485,155.557
C00698=1066.925,236.603,412.838,173.494,30.481,155.557
C00699=1066.921,236.386,412.861,173.492,30.478,155.556
C00700=1066.915,236.168,412.884,173.490,30.474,155.555
C00701=1066.910,235.951,412.908,173.489,30.471,155.555
C00702=1066.905,235.733,412.932,173.486,30.467,155.554
C00703=1066.900,235.516,412.955,173.484,30.463,155.554
C00704=1066.894,235.298,412.979,173.482,30.460,155.553
C00705=1066.889,235.080,413.003,173.481,30.457,155.552
C00706=1066.884,234.863,413.026,173.478,30.453,155.552
C00707=1066.878,234.615,413.054,173.476,30.449,155.551
C00708=1066.872,234.366,413.081,173.474,30.445,155.550
C00709=1066.866,234.118,413.107,173.472,30.441,155.550
C00710=1066.860,233.870,413.134,173.469,30.437,155.549
C00711=1066.855,233.621,413.161,173.467,30.433,155.548
C00712=1066.848,233.372,413.188,173.465,30.429,155.548
C00713=1066.842,233.124,413.215,173.462,30.425,155.547
C00714=1066.836,232.876,413.242,173.461,30.421,155.546
C00715=1066.830,232.627,413.269,173.458,30.417,155.546
C00716=1066.824,232.379,413.295,173.456,30.413,155.545
C00717=1066.818,232.130,413.322,173.454,30.409,155.544
C00718=1066.813,231.882,413.349,173.452,30.405,155.543
C00719=1066.806,231.633,413.376,173.450,30.401,155.543
C00720=1066.800,231.384,413.402,173.448,30.397,155.542
C00721=1066.795,231.136,413.429,173.445,30.393,155.541
C00722=1066.789,230.888,413.456,173.443,30.389,155.541
C00723=1066.783,230.639,413.483,173.441,30.385,155.540
C00724=1066.777,230.390,413.509,173.438,30.381,155.539
C00725=1066.771,230.142,413.536,173.437,30.377,155.538
C00726=1066.765,229.894,413.563,173.434,30.373,155.538
C00727=1066.759,229.645,413.589,173.432,30.369,155.537
C00728=1066.753,229.396,413.616,173.430,30.365,155.536
C00729=1066.748,229.147,413.642,173.428,30.361,155.536
C00730=1066.742,228.899,413.669,173.425,30.357,155.535
C00731=1066.735,228.650,413.695,173.424,30.353,155.534
C00732=1066.729,228.402,413.722,173.421,30.349,155.534
C00733=1066.723,228.153,413.749,173.419,30.345,155.533
C00734=1066.717,227.905,413.775,173.417,30.341,155.532
C00735=1066.711,227.657,413.801,173.415,30.337,155.532
C00736=1066.705,227.407,413.828,173.413,30.333,155.531
C00737=1066.699,227.159,413.854,173.411,30.329,155.530
C00738=1066.693,226.911,413.881,173.408,30.325,155.530
C00739=1066.687,226.662,413.907,173.407,30.321,155.529
C00740=1066.681,226.414,413.934,173.404,30.317,155.528
C00741=1066.675,226.165,413.959,173.402,30.314,155.528
C00742=1066.669,225.916,413.986,173.400,30.309,155.527
C00743=1066.663,225.668,414.013,173.398,30.305,155.526
C00744=1066.657,225.419,414.038,173.395,30.301,155.525
C00745=1066.651,225.171,414.065,173.394,30.297,155.525
C00746=1066.646,224.922,414.092,173.391,30.293,155.524
C00747=1066.639,224.674,414.118,173.389,30.289,155.523
C00748=1066.634,224.425,414.144,173.387,30.285,155.523
C00749=1066.628,224.177,414.170,173.385,30.281,155.522
C00750=1066.621,223.928,414.197,173.383,30.277,155.521
C00751=1066.615,223.679,414.223,173.381,30.273,155.520
C00752=1066.609,223.431,414.249,173.378,30.269,155.520
C00753=1066.604,223.182,414.275,173.377,30.265,155.519
C00754=1066.598,222.934,414.302,173.374,30.261,155.518
C00755=1066.593,222.712,414.324,173.372,30.257,155.518
C00756=1066.587,222.491,414.348,173.371,30.253,155.517
C00757=1066.582,222.269,414.371,173.369,30.250,155.517
C00758=1066.577,222.048,414.394,173.366,30.246,155.516
C00759=1066.571,221.826,414.419,173.365,30.243,155.515
C00760=1066.566,221.605,414.442,173.363,30.239,155.515
C00761=1066.561,221.383,414.465,173.361,30.236,155.514
C00762=1066.556,221.161,414.488,173.360,30.232,155.513
C00763=1066.549,220.913,414.514,173.357,30.228,155.513
C00764=1066.544,220.664,414.540,173.355,30.224,155.512
C00765=1066.537,220.416,414.566,173.353,30.220,155.511
C00766=1066.532,220.167,414.592,173.351,30.216,155.511
C00767=1066.525,219.919,414.618,173.349,30.212,155.510
C00768=1066.520,219.670,414.644,173.347,30.208,155.509
C00769=1066.513,219.422,414.670,173.344,30.204,155.509
C00770=1066.508,219.173,414.696,173.343,30.200,155.508
C00771=1066.502,218.924,414.721,173.341,30.196,155.507
C00772=1066.496,218.676,414.748,173.338,30.192,155.506
C00773=1066.490,218.427,414.773,173.337,30.188,155.506
C00774=1066.483,218.179,414.799,173.334,30.184,155.505
C00775=1066.478,217.930,414.825,173.333,30.180,155.504
C00776=1066.472,217.682,414.851,173.330,30.175,155.504
C00777=1066.466,217.433,414.877,173.328,30.172,155.503
C00778=1066.460,217.185,414.903,173.327,30.167,155.502
C00779=1066.454,216.936,414.928,173.324,30.163,155.502
C00780=1066.448,216.687,414.954,173.322,30.160,155.501
C00781=1066.442,216.439,414.980,173.320,30.155,155.500
C00782=1066.436,216.190,415.006,173.318,30.151,155.499
C00783=1066.430,215.941,415.031,173.316,30.147,155.499
C00784=1066.424,215.692,415.057,173.314,30.143,155.498
C00785=1066.418,215.444,415.083,173.312,30.139,155.497
C00786=1066.412,215.195,415.109,173.310,30.135,155.497
C00787=1066.406,214.947,415.134,173.308,30.131,155.496
C00788=1066.401,214.698,415.160,173.306,30.127,155.495
C00789=1066.394,214.450,415.186,173.304,30.123,155.495
C00790=1066.388,214.201,415.212,173.301,30.118,155.494
C00791=1066.383,213.953,415.237,173.300,30.115,155.493
C00792=1066.377,213.704,415.263,173.298,30.110,155.492
C00793=1066.371,213.455,415.289,173.296,30.106,155.492
C00794=1066.365,213.206,415.314,173.294,30.102,155.491
C00795=1066.359,212.958,415.339,173.291,30.098,155.490
C00796=1066.354,212.709,415.365,173.290,30.094,155.489
C00797=1066.347,212.461,415.391,173.288,30.090,155.489
C00798=1066.341,212.212,415.417,173.285,30.086,155.488
C00799=1066.335,211.963,415.442,173.284,30.082,155.487
C00800=1066.330,211.715,415.467,173.282,30.078,155.487
C00801=1066.324,211.466,415.493,173.280,30.074,155.486
C00802=1066.317,211.218,415.518,173.278,30.070,155.485
C00803=1066.311,210.969,415.543,173.275,30.065,155.485
C00804=1066.306,210.720,415.569,173.274,30.062,155.484
C00805=1066.299,210.471,415.595,173.272,30.057,155.483
C00806=1066.293,210.223,415.620,173.270,30.053,155.482
C00807=1066.287,209.974,415.645,173.268,30.050,155.482
C00808=1066.281,209.726,415.670,173.265,30.045,155.481
C00809=1066.276,209.477,415.696,173.264,30.041,155.480
C00810=1066.270,209.228,415.722,173.262,30.037,155.480
C00811=1066.264,209.010,415.743,173.261,30.034,155.479
C00812=1066.259,208.790,415.766,173.258,30.030,155.478
C00813=1066.253,208.571,415.788,173.256,30.026,155.478
C00814=1066.249,208.352,415.810,173.255,30.022,155.477
C00815=1066.244,208.133,415.833,173.253,30.019,155.477
C00816=1066.238,207.913,415.855,173.251,30.015,155.476
C00817=1066.233,207.694,415.877,173.250,30.012,155.475
C00818=1066.228,207.475,415.899,173.248,30.008,155.475
C00819=1066.203,206.430,416.002,173.094,29.931,155.470
C00820=1066.197,206.180,416.027,173.091,29.928,155.469
C00821=1066.192,205.932,416.051,173.089,29.925,155.469
C00822=1066.186,205.683,416.075,173.087,29.922,155.468
C00823=1066.180,205.434,416.101,173.085,29.918,155.468
C00824=1066.174,205.186,416.124,173.082,29.916,155.467
C00825=1066.168,204.937,416.149,173.081,29.912,155.467
C00826=1066.163,204.688,416.173,173.078,29.909,155.466
C00827=1066.157,204.439,416.198,173.075,29.906,155.466
C00828=1066.152,204.190,416.222,173.074,29.903,155.465
C00829=1066.146,203.942,416.246,173.071,29.899,155.465
C00830=1066.140,203.693,416.270,173.069,29.896,155.464
C00831=1066.134,203.444,416.295,173.067,29.893,155.464
C00832=1066.128,203.196,416.320,173.065,29.890,155.463
C00833=1066.123,202.947,416.344,173.062,29.887,155.463
C00834=1066.117,202.699,416.368,173.061,29.884,155.462
C00835=1066.111,202.449,416.392,173.058,29.880,155.462
C00836=1066.106,202.201,416.417,173.056,29.877,155.461
C00837=1066.099,201.952,416.441,173.054,29.874,155.461
C00838=1066.094,201.703,416.465,173.052,29.871,155.460
C00839=1066.088,201.455,416.489,173.049,29.868,155.460
C00840=1066.082,201.206,416.513,173.048,29.865,155.459
C00841=1066.077,200.957,416.537,173.045,29.862,155.459
C00842=1066.070,200.708,416.561,173.042,29.858,155.458
C00843=1066.065,200.459,416.585,173.041,29.855,155.458
C00844=1066.059,200.211,416.609,173.038,29.852,155.457
C00845=1066.053,199.961,416.633,173.036,29.849,155.457
C00846=1066.047,199.713,416.657,173.034,29.846,155.457
C00847=1066.041,199.464,416.682,173.032,29.843,155.456
C00848=1066.035,199.216,416.705,173.029,29.840,155.456
C00849=1066.030,198.967,416.730,173.028,29.837,155.455
C00850=1066.023,198.717,416.753,173.025,29.834,155.455
C00851=1066.018,198.469,416.777,173.023,29.831,155.454
C00852=1066.012,198.221,416.801,173.021,29.828,155.454
C00853=1066.005,197.972,416.825,173.019,29.825,155.453
C00854=1066.000,197.723,416.849,173.016,29.821,155.453
C00855=1065.994,197.475,416.873,173.015,29.819,155.452
C00856=1065.988,197.225,416.897,173.012,29.815,155.452
C00857=1065.982,196.977,416.920,173.010,29.813,155.451
C00858=1065.977,196.728,416.945,173.008,29.809,155.451
C00859=1065.970,196.479,416.969,173.006,29.806,155.450
C00860=1065.965,196.230,416.992,173.003,29.803,155.450
C00861=1065.959,195.981,417.016,173.002,29.800,155.449
C00862=1065.954,195.732,417.040,172.999,29.797,155.449
C00863=1065.948,195.483,417.063,172.997,29.794,155.448
C00864=1065.943,195.235,417.088,172.996,29.791,155.448
C00865=1065.936,194.986,417.111,172.993,29.788,155.448
C00866=1065.930,194.737,417.135,172.991,29.785,155.447
C00867=1065.925,194.488,417.159,172.989,29.782,155.447
C00868=1065.919,194.240,417.182,172.987,29.778,155.446
C00869=1065.914,193.991,417.206,172.984,29.776,155.446
C00870=1065.907,193.742,417.230,172.983,29.772,155.445
C00871=1065.902,193.493,417.254,172.980,29.769,155.445
C00872=1065.896,193.244,417.277,172.978,29.766,155.444
C00873=1065.890,192.996,417.301,172.976,29.763,155.444
C00874=1065.885,192.747,417.324,172.974,29.760,155.443
C00875=1065.878,192.498,417.348,172.972,29.757,155.443
C00876=1065.873,192.249,417.373,172.970,29.754,155.442
C00877=1065.867,192.000,417.396,172.968,29.751,155.442
C00878=1065.861,191.752,417.419,172.965,29.748,155.441
C00879=1065.856,191.503,417.443,172.964,29.745,155.441
C00880=1065.850,191.220,417.470,172.961,29.741,155.440
C00881=1065.843,190.938,417.497,172.959,29.738,155.440
C00882=1065.836,190.655,417.524,172.957,29.735,155.439
C00883=1065.830,190.372,417.550,172.954,29.731,155.439
C00884=1065.825,190.123,417.574,172.952,29.728,155.438
C00885=1065.819,189.874,417.597,172.950,29.725,155.438
C00886=1065.813,189.625,417.622,172.948,29.722,155.437
C00887=1065.807,189.376,417.645,172.946,29.719,155.437
C00888=1065.801,189.128,417.668,172.944,29.716,155.436
C00889=1065.796,188.879,417.692,172.941,29.712,155.436
C00890=1065.790,188.630,417.715,172.940,29.710,155.436
C00891=1065.784,188.382,417.738,172.937,29.706,155.435
C00892=1065.779,188.132,417.762,172.935,29.704,155.435
C00893=1065.773,187.884,417.786,172.934,29.700,155.434
C00894=1065.768,187.635,417.808,172.931,29.697,155.434
C00895=1065.763,187.386,417.832,172.929,29.694,155.433
C00896=1065.756,187.137,417.856,172.927,29.691,155.433
C00897=1065.750,186.888,417.879,172.925,29.688,155.432
C00898=1065.745,186.639,417.903,172.923,29.685,155.432
C00899=1065.739,186.391,417.926,172.921,29.682,155.431
C00900=1065.734,186.142,417.949,172.919,29.679,155.431
C00901=1065.729,185.893,417.973,172.917,29.676,155.430
C00902=1065.723,185.644,417.996,172.915,29.673,155.430
C00903=1065.717,185.395,418.019,172.913,29.670,155.429
C00904=1065.712,185.146,418.043,172.911,29.666,155.429
C00905=1065.706,184.897,418.066,172.909,29.664,155.428
C00906=1065.700,184.648,418.089,172.907,29.661,155.428
C00907=1065.694,184.400,418.112,172.905,29.658,155.428
C00908=1065.689,184.151,418.135,172.903,29.655,155.427
C00909=1065.683,183.902,418.158,172.901,29.652,155.427
C00910=1065.676,183.653,418.182,172.899,29.649,155.426
C00911=1065.671,183.404,418.205,172.897,29.646,155.426
C00912=1065.665,183.155,418.227,172.894,29.643,155.425
C00913=1065.659,182.907,418.251,172.893,29.640,155.425
C00914=1065.653,182.658,418.274,172.891,29.637,155.424
C00915=1065.647,182.409,418.296,172.888,29.635,155.424
C00916=1065.641,182.160,418.319,172.886,29.632,155.424
C00917=1065.635,181.911,418.342,172.885,29.629,155.423
C00918=1065.629,181.662,418.366,172.882,29.626,155.423
C00919=1065.623,181.413,418.389,172.880,29.623,155.422
C00920=1065.618,181.164,418.412,172.878,29.620,155.422
C00921=1065.612,180.915,418.434,172.876,29.617,155.421
C00922=1065.605,180.667,418.457,172.874,29.614,155.421
C00923=1065.600,180.418,418.480,172.872,29.611,155.421
C00924=1065.594,180.169,418.503,172.870,29.609,155.420
C00925=1065.588,179.920,418.526,172.868,29.605,155.420
C00926=1065.582,179.671,418.549,172.866,29.603,155.419
C00927=1065.577,179.422,418.572,172.864,29.600,155.419
C00928=1065.570,179.173,418.594,172.862,29.597,155.418
C00929=1065.564,178.925,418.617,172.860,29.594,155.418
C00930=1065.559,178.676,418.640,172.858,29.591,155.418
C00931=1065.553,178.427,418.663,172.856,29.588,155.417
C00932=1065.547,178.178,418.686,172.854,29.585,155.417
C00933=1065.541,177.929,418.708,172.852,29.582,155.416
C00934=1065.535,177.680,418.731,172.850,29.580,155.416
C00935=1065.529,177.431,418.754,172.848,29.577,155.415
C00936=1065.524,177.183,418.777,172.846,29.573,155.415
C00937=1065.518,176.933,418.799,172.844,29.571,155.414
C00938=1065.512,176.684,418.822,172.842,29.568,155.414
C00939=1065.506,176.436,418.844,172.840,29.565,155.414
C00940=1065.500,176.187,418.867,172.839,29.562,155.413
C00941=1065.495,175.938,418.890,172.836,29.559,155.413
C00942=1065.489,175.689,418.913,172.834,29.556,155.412
C00943=1065.482,175.440,418.936,172.833,29.553,155.412
C00944=1065.476,175.157,418.961,172.830,29.550,155.411
C00945=1065.469,174.873,418.987,172.828,29.547,155.411
C00946=1065.463,174.590,419.013,172.826,29.543,155.410
C00947=1065.457,174.308,419.039,172.823,29.540,155.410
C00948=1065.451,174.058,419.061,172.821,29.537,155.409
C00949=1065.445,173.810,419.083,172.820,29.534,155.409
C00950=1065.439,173.561,419.106,172.817,29.531,155.409
C00951=1065.434,173.312,419.129,172.815,29.528,155.408
C00952=1065.428,173.063,419.151,172.814,29.526,155.408
C00953=1065.422,172.814,419.174,172.812,29.523,155.407
C00954=1065.416,172.565,419.197,172.809,29.520,155.407
C00955=1065.410,172.316,419.220,172.808,29.517,155.406
C00956=1065.405,172.067,419.241,172.806,29.514,155.406
C00957=1065.399,171.819,419.264,172.803,29.511,155.405
C00958=1065.393,171.570,419.287,172.802,29.508,155.405
C00959=1065.388,171.320,419.309,172.800,29.505,155.405
C00960=1065.382,171.071,419.332,172.798,29.502,155.404
C00961=1065.376,170.823,419.354,172.796,29.499,155.404
C00962=1065.370,170.573,419.376,172.794,29.497,155.403
C00963=1065.365,170.325,419.399,172.792,29.494,155.403
C00964=1065.359,170.076,419.421,172.791,29.491,155.402
C00965=1065.353,169.827,419.444,172.788,29.488,155.402
C00966=1065.347,169.578,419.467,172.787,29.485,155.402
C00967=1065.342,169.329,419.489,172.785,29.482,155.401
C00968=1065.336,169.081,419.511,172.783,29.479,155.401
C00969=1065.331,168.831,419.533,172.781,29.476,155.400
C00970=1065.325,168.582,419.556,172.779,29.473,155.400
C00971=1065.319,168.333,419.578,172.777,29.470,155.399
C00972=1065.313,168.084,419.601,172.776,29.468,155.399
C00973=1065.308,167.835,419.622,172.773,29.465,155.398
C00974=1065.302,167.587,419.645,172.771,29.461,155.398
C00975=1065.296,167.337,419.667,172.770,29.459,155.398
C00976=1065.291,167.088,419.690,172.768,29.456,155.397
C00977=1065.286,166.840,419.712,172.765,29.453,155.397
C00978=1065.279,166.591,419.734,172.764,29.450,155.396
C00979=1065.274,166.342,419.756,172.762,29.447,155.396
C00980=1065.268,166.093,419.779,172.760,29.444,155.395
C00981=1065.263,165.844,419.801,172.758,29.441,155.395
C00982=1065.257,165.595,419.824,172.756,29.438,155.394
C00983=1065.251,165.346,419.846,172.754,29.435,155.394
C00984=1065.246,165.097,419.867,172.753,29.432,155.394
C00985=1065.240,164.848,419.890,172.751,29.430,155.393
C00986=1065.235,164.599,419.912,172.748,29.427,155.393
C00987=1065.229,164.351,419.934,172.747,29.423,155.392
C00988=1065.223,164.101,419.956,172.745,29.421,155.392
C00989=1065.218,163.852,419.979,172.743,29.418,155.391
C00990=1065.212,163.604,420.001,172.741,29.415,155.391
C00991=1065.207,163.354,420.023,172.739,29.412,155.390
C00992=1065.200,163.105,420.045,172.738,29.409,155.390
C00993=1065.195,162.857,420.067,172.736,29.406,155.390
C00994=1065.190,162.608,420.089,172.734,29.403,155.389
C00995=1065.184,162.358,420.111,172.732,29.400,155.389
C00996=1065.179,162.110,420.134,172.730,29.397,155.388
C00997=1065.173,161.861,420.156,172.728,29.394,155.388
C00998=1065.167,161.611,420.177,172.727,29.392,155.387
C00999=1065.162,161.363,420.200,172.725,29.388,155.387
C01000=1065.156,161.114,420.222,172.723,29.386,155.386
C01001=1065.150,160.864,420.244,172.721,29.383,155.386
C01002=1065.145,160.616,420.265,172.719,29.380,155.386
C01003=1065.139,160.367,420.287,172.717,29.377,155.385
C01004=1065.133,160.118,420.310,172.716,29.374,155.385
C01005=1065.127,159.869,420.331,172.714,29.371,155.384
C01006=1065.121,159.620,420.353,172.711,29.368,155.384
C01007=1065.116,159.371,420.375,172.710,29.366,155.383
C01008=1065.109,159.087,420.400,172.708,29.363,155.383
C01009=1065.102,158.805,420.424,172.706,29.360,155.383
C01010=1065.096,158.521,420.449,172.704,29.356,155.382
C01011=1065.089,158.237,420.474,172.701,29.353,155.382
C01012=1065.083,157.988,420.496,172.700,29.350,155.381
C01013=1065.078,157.739,420.517,172.698,29.347,155.381
C01014=1065.072,157.490,420.539,172.696,29.345,155.380
C01015=1065.066,157.241,420.561,172.694,29.342,155.380
C01016=1065.061,156.992,420.583,172.692,29.339,155.379
C01017=1065.055,156.743,420.604,172.690,29.336,155.379
C01018=1065.049,156.494,420.626,172.689,29.333,155.379
C01019=1065.043,156.245,420.647,172.687,29.330,155.378
C01020=1065.038,155.996,420.669,172.685,29.328,155.378
C01021=1065.032,155.747,420.691,172.683,29.325,155.377
C01022=1065.026,155.498,420.712,172.681,29.322,155.377
C01023=1065.020,155.249,420.734,172.680,29.319,155.376
C01024=1065.014,155.000,420.755,172.678,29.316,155.376
C01025=1065.009,154.751,420.777,172.676,29.313,155.376
C01026=1065.003,154.502,420.799,172.675,29.311,155.375
C01027=1064.997,154.253,420.820,172.672,29.308,155.375
C01028=1064.991,154.004,420.842,172.670,29.305,155.374
C01029=1064.985,153.755,420.863,172.669,29.302,155.374
C01030=1064.979,153.506,420.885,172.667,29.300,155.374
C01031=1064.973,153.258,420.906,172.665,29.296,155.373
C01032=1064.968,153.008,420.928,172.664,29.294,155.373
C01033=1064.962,152.759,420.950,172.662,29.291,155.372
C01034=1064.956,152.510,420.971,172.659,29.288,155.372
C01035=1064.950,152.261,420.993,172.658,29.285,155.371
C01036=1064.945,152.012,421.013,172.656,29.283,155.371
C01037=1064.939,151.763,421.035,172.654,29.280,155.371
C01038=1064.933,151.514,421.056,172.653,29.277,155.370
C01039=1064.927,151.265,421.078,172.651,29.274,155.370
C01040=1064.922,151.016,421.100,172.649,29.271,155.369
C01041=1064.916,150.767,421.121,172.647,29.268,155.369
C01042=1064.910,150.517,421.142,172.645,29.266,155.369
C01043=1064.905,150.269,421.164,172.643,29.263,155.368
C01044=1064.898,150.020,421.185,172.642,29.260,155.368
C01045=1064.893,149.771,421.207,172.640,29.257,155.367
C01046=1064.887,149.522,421.228,172.638,29.255,155.367
C01047=1064.881,149.273,421.249,172.637,29.251,155.366
C01048=1064.875,149.024,421.270,172.635,29.249,155.366
C01049=1064.870,148.775,421.292,172.633,29.246,155.366
C01050=1064.864,148.526,421.313,172.631,29.243,155.365
C01051=1064.858,148.277,421.334,172.629,29.240,155.365
C01052=1064.852,148.028,421.355,172.628,29.238,155.364
C01053=1064.847,147.779,421.377,172.626,29.235,155.364
C01054=1064.841,147.529,421.398,172.624,29.232,155.364
C01055=1064.835,147.281,421.419,172.623,29.230,155.363
C01056=1064.829,147.031,421.441,172.621,29.227,155.363
C01057=1064.823,146.783,421.462,172.618,29.224,155.362
C01058=1064.817,146.533,421.482,172.617,29.221,155.362
C01059=1064.811,146.285,421.503,172.615,29.218,155.361
C01060=1064.805,146.035,421.524,172.613,29.215,155.361
C01061=1064.800,145.787,421.546,172.612,29.212,155.361
C01062=1064.794,145.537,421.567,172.610,29.210,155.360
C01063=1064.788,145.288,421.588,172.608,29.207,155.360
C01064=1064.782,145.039,421.609,172.607,29.204,155.359
C01065=1064.777,144.790,421.630,172.605,29.202,155.359
C01066=1064.770,144.541,421.651,172.603,29.199,155.359
C01067=1064.765,144.293,421.672,172.601,29.196,155.358
C01068=1064.759,144.043,421.693,172.599,29.193,155.358
C01069=1064.753,143.794,421.715,172.598,29.191,155.357
C01070=1064.748,143.545,421.735,172.596,29.188,155.357
C01071=1064.742,143.296,421.757,172.594,29.185,155.357
C01072=1064.735,143.012,421.781,172.593,29.182,155.356
C01073=1064.729,142.729,421.804,172.590,29.178,155.355
C01074=1064.722,142.444,421.828,172.588,29.176,155.355
C01075=1064.715,142.160,421.852,172.587,29.172,155.355
C01076=1064.709,141.912,421.873,172.584,29.169,155.354
C01077=1064.704,141.663,421.894,172.583,29.167,155.354
C01078=1064.698,141.414,421.915,172.581,29.164,155.353
C01079=1064.692,141.165,421.936,172.579,29.161,155.353
C01080=1064.687,140.915,421.957,172.578,29.159,155.353
C01081=1064.680,140.667,421.977,172.576,29.156,155.352
C01082=1064.675,140.418,421.998,172.574,29.153,155.352
C01083=1064.669,140.168,422.020,172.573,29.150,155.351
C01084=1064.664,139.919,422.040,172.571,29.147,155.351
C01085=1064.658,139.670,422.062,172.569,29.144,155.350
C01086=1064.652,139.421,422.082,172.568,29.142,155.350
C01087=1064.646,139.172,422.102,172.566,29.139,155.350
C01088=1064.640,138.923,422.124,172.565,29.136,155.349
C01089=1064.634,138.674,422.144,172.562,29.133,155.349
C01090=1064.629,138.425,422.164,172.560,29.131,155.348
C01091=1064.623,138.176,422.186,172.559,29.128,155.348
C01092=1064.617,137.927,422.206,172.557,29.125,155.348
C01093=1064.611,137.677,422.227,172.555,29.122,155.347
C01094=1064.605,137.429,422.248,172.554,29.120,155.347
C01095=1064.599,137.180,422.268,172.552,29.117,155.346
C01096=1064.593,136.930,422.289,172.550,29.114,155.346
C01097=1064.587,136.682,422.310,172.549,29.111,155.346
C01098=1064.582,136.433,422.330,172.547,29.109,155.345
C01099=1064.576,136.183,422.351,172.545,29.106,155.345
C01100=1064.570,135.934,422.371,172.544,29.103,155.344
C01101=1064.564,135.686,422.392,172.542,29.101,155.344
C01102=1064.558,135.436,422.413,172.540,29.098,155.343
C01103=1064.553,135.187,422.433,172.539,29.095,155.343
C01104=1064.547,134.938,422.454,172.537,29.092,155.343
C01105=1064.541,134.688,422.474,172.536,29.090,155.342
C01106=1064.535,134.440,422.495,172.534,29.087,155.342
C01107=1064.529,134.191,422.515,172.531,29.084,155.341
C01108=1064.523,133.941,422.536,172.530,29.081,155.341
C01109=1064.518,133.692,422.557,172.528,29.079,155.341
C01110=1064.512,133.443,422.577,172.526,29.076,155.340
C01111=1064.507,133.195,422.598,172.525,29.073,155.340
C01112=1064.500,132.945,422.618,172.523,29.070,155.339
C01113=1064.495,132.696,422.639,172.521,29.067,155.339
C01114=1064.489,132.447,422.659,172.520,29.064,155.339
C01115=1064.483,132.198,422.680,172.518,29.062,155.338
C01116=1064.478,131.948,422.700,172.517,29.059,155.338
C01117=1064.472,131.699,422.720,172.515,29.056,155.337
C01118=1064.466,131.451,422.740,172.513,29.053,155.337
C01119=1064.460,131.201,422.761,172.512,29.051,155.336
C01120=1064.453,130.953,422.782,172.510,29.048,155.336
C01121=1064.447,130.704,422.802,172.508,29.046,155.336
C01122=1064.442,130.454,422.823,172.507,29.043,155.335
C01123=1064.436,130.205,422.843,172.505,29.040,155.335
C01124=1064.430,129.956,422.863,172.503,29.038,155.335
C01125=1064.424,129.707,422.883,172.502,29.035,155.334
C01126=1064.418,129.458,422.904,172.500,29.032,155.334
C01127=1064.412,129.209,422.924,172.498,29.029,155.333
C01128=1064.406,128.960,422.944,172.497,29.027,155.333
C01129=1064.400,128.710,422.964,172.495,29.024,155.333
C01130=1064.394,128.461,422.984,172.493,29.021,155.332
C01131=1064.388,128.213,423.004,172.492,29.019,155.332
C01132=1064.383,127.964,423.025,172.490,29.016,155.331
C01133=1064.376,127.713,423.045,172.489,29.013,155.331
C01134=1064.370,127.465,423.064,172.487,29.010,155.331
C01135=1064.365,127.215,423.085,172.485,29.008,155.330
C01136=1064.358,126.932,423.108,172.483,29.005,155.330
C01137=1064.351,126.648,423.131,172.481,29.001,155.329
C01138=1064.345,126.363,423.154,172.479,28.999,155.329
C01139=1064.338,126.080,423.177,172.477,28.995,155.328
C01140=1064.332,125.832,423.197,172.475,28.992,155.328
C01141=1064.326,125.581,423.217,172.474,28.990,155.328
C01142=1064.320,125.332,423.237,172.472,28.987,155.327
C01143=1064.314,125.083,423.257,172.470,28.984,155.327
C01144=1064.308,124.835,423.277,172.469,28.981,155.326
C01145=1064.302,124.586,423.297,172.467,28.979,155.326
C01146=1064.296,124.336,423.318,172.465,28.976,155.325
C01147=1064.290,124.087,423.338,172.464,28.973,155.325
C01148=1064.285,123.838,423.357,172.462,28.970,155.325
C01149=1064.279,123.589,423.377,172.460,28.968,155.324
C01150=1064.274,123.340,423.398,172.459,28.966,155.324
C01151=1064.268,123.091,423.418,172.457,28.963,155.324
C01152=1064.262,122.842,423.438,172.456,28.960,155.323
C01153=1064.255,122.592,423.457,172.454,28.957,155.323
C01154=1064.250,122.343,423.478,172.453,28.955,155.322
C01155=1064.244,122.094,423.498,172.452,28.952,155.322
C01156=1064.238,121.845,423.518,172.450,28.949,155.322
C01157=1064.232,121.596,423.537,172.448,28.946,155.321
C01158=1064.227,121.347,423.558,172.447,28.943,155.321
C01159=1064.221,121.098,423.577,172.445,28.941,155.320
C01160=1064.215,120.849,423.597,172.444,28.938,155.320
C01161=1064.209,120.599,423.617,172.442,28.935,155.319
C01162=1064.203,120.350,423.637,172.440,28.932,155.319
C01163=1064.198,120.100,423.657,172.439,28.930,155.319
C01164=1064.192,119.852,423.677,172.437,28.927,155.318
C01165=1064.186,119.603,423.697,172.435,28.924,155.318
C01166=1064.180,119.353,423.716,172.434,28.921,155.317
C01167=1064.174,119.105,423.736,172.432,28.919,155.317
C01168=1064.169,118.855,423.757,172.430,28.916,155.317
C01169=1064.163,118.606,423.776,172.429,28.913,155.316
C01170=1064.157,118.357,423.796,172.427,28.910,155.316
C01171=1064.151,118.108,423.816,172.426,28.908,155.315
C01172=1064.146,117.859,423.835,172.424,28.905,155.315
C01173=1064.140,117.610,423.855,172.422,28.902,155.315
C01174=1064.135,117.360,423.875,172.421,28.899,155.314
C01175=1064.129,117.112,423.895,172.419,28.897,155.314
C01176=1064.122,116.862,423.915,172.417,28.894,155.313
C01177=1064.116,116.613,423.934,172.416,28.891,155.313
C01178=1064.110,116.364,423.954,172.414,28.889,155.312
C01179=1064.105,116.114,423.974,172.413,28.886,155.312
C01180=1064.099,115.865,423.994,172.411,28.883,155.312
C01181=1064.094,115.616,424.013,172.409,28.880,155.311
C01182=1064.088,115.367,424.033,172.408,28.877,155.311
C01183=1064.082,115.118,424.052,172.406,28.874,155.310
C01184=1064.076,114.869,424.072,172.404,28.871,155.310
C01185=1064.071,114.619,424.092,172.404,28.869,155.310
C01186=1064.065,114.370,424.112,172.402,28.866,155.309
C01187=1064.059,114.121,424.131,172.401,28.863,155.309
C01188=1064.053,113.872,424.151,172.399,28.861,155.308
C01189=1064.048,113.623,424.171,172.397,28.858,155.308
C01190=1064.042,113.374,424.191,172.396,28.855,155.307
C01191=1064.036,113.124,424.210,172.394,28.852,155.307
C01192=1064.030,112.875,424.229,172.392,28.850,155.307
C01193=1064.024,112.626,424.249,172.391,28.847,155.306
C01194=1064.018,112.377,424.268,172.389,28.844,155.306
C01195=1064.012,112.128,424.288,172.388,28.842,155.305
C01196=1064.006,111.879,424.307,172.386,28.839,155.305
C01197=1064.001,111.629,424.326,172.384,28.836,155.305
C01198=1063.995,111.380,424.346,172.383,28.833,155.304
C01199=1063.989,111.131,424.365,172.381,28.831,155.304
C01200=1063.982,110.847,424.388,172.379,28.828,155.303
C01201=1063.976,110.564,424.410,172.378,28.825,155.303
C01202=1063.968,110.279,424.431,172.376,28.822,155.303
C01203=1063.962,109.995,424.454,172.374,28.819,155.302
C01204=1063.956,109.746,424.473,172.372,28.816,155.302
C01205=1063.950,109.497,424.492,172.370,28.813,155.301
C01206=1063.944,109.248,424.512,172.370,28.811,155.301
C01207=1063.938,108.999,424.531,172.368,28.808,155.301
C01208=1063.932,108.749,424.550,172.366,28.805,155.300
C01209=1063.926,108.500,424.570,172.365,28.802,155.300
C01210=1063.920,108.251,424.589,172.363,28.800,155.299
C01211=1063.915,108.001,424.609,172.362,28.797,155.299
C01212=1063.908,107.752,424.627,172.360,28.794,155.299
C01213=1063.903,107.503,424.646,172.358,28.791,155.298
C01214=1063.897,107.254,424.666,172.357,28.789,155.298
C01215=1063.892,107.005,424.685,172.355,28.786,155.297
C01216=1063.885,106.756,424.704,172.354,28.783,155.297
C01217=1063.879,106.507,424.723,172.352,28.780,155.297
C01218=1063.874,106.257,424.742,172.350,28.778,155.296
C01219=1063.868,106.009,424.762,172.349,28.776,155.296
C01220=1063.861,105.759,424.781,172.347,28.773,155.295
C01221=1063.856,105.510,424.800,172.346,28.770,155.295
C01222=1063.850,105.261,424.819,172.345,28.768,155.295
C01223=1063.844,105.011,424.839,172.343,28.765,155.294
C01224=1063.838,104.762,424.857,172.341,28.762,155.294
C01225=1063.832,104.513,424.877,172.340,28.759,155.293
C01226=1063.826,104.264,424.897,172.338,28.757,155.293
C01227=1063.821,104.015,424.915,172.337,28.754,155.293
C01228=1063.815,103.766,424.934,172.335,28.751,155.292
C01229=1063.809,103.517,424.953,172.333,28.748,155.292
C01230=1063.803,103.267,424.973,172.332,28.745,155.291
C01231=1063.798,103.018,424.992,172.330,28.743,155.291
C01232=1063.791,102.769,425.010,172.329,28.740,155.291
C01233=1063.786,102.519,425.030,172.327,28.737,155.290
C01234=1063.780,102.270,425.049,172.326,28.735,155.290
C01235=1063.775,102.021,425.068,172.325,28.732,155.289
C01236=1063.768,101.772,425.086,172.323,28.729,155.289
C01237=1063.763,101.522,425.106,172.321,28.726,155.289
C01238=1063.757,101.274,425.126,172.320,28.724,155.288
C01239=1063.750,101.024,425.144,172.318,28.721,155.288
C01240=1063.745,100.776,425.163,172.317,28.718,155.287
C01241=1063.739,100.526,425.181,172.315,28.715,155.287
C01242=1063.733,100.277,425.200,172.313,28.713,155.287
C01243=1063.727,100.027,425.219,172.312,28.710,155.286
C01244=1063.721,99.778,425.238,172.310,28.707,155.286
C01245=1063.715,99.529,425.257,172.309,28.705,155.285
C01246=1063.709,99.279,425.276,172.308,28.702,155.285
C01247=1063.703,99.030,425.295,172.306,28.700,155.285
C01248=1063.698,98.782,425.314,172.305,28.697,155.284
C01249=1063.691,98.532,425.332,172.303,28.694,155.284
C01250=1063.685,98.283,425.352,172.301,28.691,155.283
C01251=1063.679,98.034,425.370,172.300,28.689,155.283
C01252=1063.673,97.784,425.389,172.298,28.686,155.283
C01253=1063.667,97.535,425.408,172.297,28.683,155.282
C01254=1063.662,97.286,425.426,172.295,28.680,155.282
C01255=1063.656,97.037,425.445,172.293,28.678,155.281
C01256=1063.650,96.787,425.464,172.293,28.675,155.281
C01257=1063.644,96.538,425.483,172.291,28.673,155.281
C01258=1063.638,96.289,425.502,172.289,28.670,155.280
C01259=1063.632,96.040,425.520,172.288,28.667,155.280
C01260=1063.626,95.791,425.540,172.286,28.665,155.279
C01261=1063.620,95.541,425.558,172.285,28.662,155.279
C01262=1063.615,95.292,425.577,172.283,28.659,155.279
C01263=1063.608,95.043,425.595,172.281,28.656,155.278
C01264=1063.600,94.676,425.623,172.279,28.652,155.278
C01265=1063.591,94.310,425.650,172.277,28.648,155.277
C01266=1063.582,93.943,425.678,172.275,28.644,155.276
C01267=1063.574,93.577,425.705,172.273,28.641,155.276
C01268=1063.568,93.328,425.723,172.271,28.638,155.276
C01269=1063.563,93.079,425.743,172.269,28.635,155.275
C01270=1063.556,92.830,425.761,172.268,28.632,155.275
C01271=1063.550,92.580,425.779,172.267,28.630,155.274
C01272=1063.545,92.331,425.798,172.265,28.627,155.274
C01273=1063.539,92.082,425.817,172.264,28.624,155.273
C01274=1063.533,91.833,425.836,172.262,28.621,155.273
C01275=1063.527,91.584,425.854,172.261,28.619,155.273
C01276=1063.522,91.334,425.873,172.259,28.616,155.272
C01277=1063.515,91.085,425.891,172.257,28.613,155.272
C01278=1063.509,90.835,425.909,172.256,28.610,155.271
C01279=1063.504,90.587,425.928,172.254,28.608,155.271
C01280=1063.498,90.337,425.946,172.254,28.605,155.271
C01281=1063.492,90.088,425.965,172.252,28.602,155.270
C01282=1063.485,89.839,425.983,172.250,28.600,155.270
C01283=1063.480,89.589,426.002,172.249,28.597,155.270
C01284=1063.474,89.340,426.020,172.247,28.595,155.269
C01285=1063.468,89.090,426.038,172.245,28.592,155.269
C01286=1063.461,88.841,426.057,172.244,28.589,155.268
C01287=1063.456,88.593,426.075,172.242,28.586,155.268
C01288=1063.450,88.343,426.094,172.241,28.584,155.268
C01289=1063.444,88.094,426.112,172.240,28.582,155.267
C01290=1063.438,87.845,426.130,172.238,28.579,155.267
C01291=1063.432,87.596,426.149,172.237,28.576,155.266
C01292=1063.426,87.346,426.166,172.235,28.573,155.266
C01293=1063.419,87.097,426.185,172.234,28.570,155.266
C01294=1063.414,86.847,426.203,172.232,28.568,155.265
C01295=1063.408,86.598,426.222,172.230,28.565,155.265
C01296=1063.402,86.348,426.240,172.229,28.562,155.264
C01297=1063.396,86.100,426.258,172.228,28.560,155.264
C01298=1063.390,85.850,426.276,172.226,28.557,155.264
C01299=1063.384,85.601,426.295,172.225,28.555,155.263
C01300=1063.379,85.352,426.313,172.223,28.552,155.263
C01301=1063.372,85.103,426.332,172.222,28.549,155.263
C01302=1063.366,84.853,426.349,172.220,28.546,155.262
C01303=1063.360,84.605,426.368,172.218,28.544,155.262
C01304=1063.354,84.355,426.386,172.217,28.541,155.261
C01305=1063.348,84.106,426.404,172.216,28.538,155.261
C01306=1063.343,83.856,426.422,172.215,28.536,155.261
C01307=1063.337,83.607,426.440,172.213,28.533,155.260
C01308=1063.327,83.191,426.471,172.211,28.529,155.260
C01309=1063.317,82.775,426.501,172.208,28.524,155.259
C01310=1063.307,82.359,426.531,172.205,28.519,155.258
C01311=1063.297,81.943,426.561,172.203,28.515,155.258
C01312=1063.291,81.693,426.579,172.201,28.512,155.257
C01313=1063.285,81.445,426.598,172.200,28.509,155.257
C01314=1063.279,81.195,426.616,172.199,28.507,155.256
C01315=1063.274,80.945,426.634,172.197,28.504,155.256
C01316=1063.268,80.697,426.652,172.196,28.502,155.256
C01317=1063.262,80.447,426.670,172.194,28.499,155.255
C01318=1063.257,80.198,426.688,172.192,28.496,155.255
C01319=1063.250,79.948,426.706,172.191,28.493,155.254
C01320=1063.245,79.700,426.724,172.190,28.491,155.254
C01321=1063.238,79.450,426.742,172.189,28.488,155.254
C01322=1063.233,79.201,426.760,172.187,28.485,155.253
C01323=1063.227,78.952,426.778,172.185,28.482,155.253
C01324=1063.220,78.667,426.799,172.184,28.480,155.252
C01325=1063.213,78.384,426.819,172.182,28.476,155.252
C01326=1063.207,78.100,426.840,172.181,28.474,155.251
C01327=1063.200,77.816,426.861,172.178,28.470,155.251
C01328=1063.194,77.567,426.878,172.178,28.467,155.251
C01329=1063.188,77.317,426.896,172.176,28.465,155.250
C01330=1063.182,77.068,426.913,172.174,28.462,155.250
C01331=1063.176,76.818,426.931,172.173,28.460,155.249
C01332=1063.170,76.570,426.949,172.171,28.457,155.249
C01333=1063.164,76.320,426.967,172.170,28.454,155.249
C01334=1063.158,76.070,426.985,172.168,28.451,155.248
C01335=1063.152,75.821,427.003,172.167,28.449,155.248
C01336=1063.146,75.572,427.021,172.166,28.447,155.248
C01337=1063.141,75.323,427.038,172.164,28.444,155.247
C01338=1063.134,75.073,427.056,172.162,28.441,155.247
C01339=1063.128,74.825,427.074,172.161,28.438,155.246
C01340=1063.122,74.575,427.092,172.159,28.436,155.246
C01341=1063.116,74.326,427.109,172.158,28.433,155.246
C01342=1063.110,74.076,427.127,172.157,28.430,155.245
C01343=1063.105,73.827,427.145,172.155,28.427,155.245
C01344=1063.098,73.577,427.163,172.154,28.425,155.244
C01345=1063.093,73.328,427.180,172.152,28.422,155.244
C01346=1063.086,73.079,427.198,172.151,28.420,155.244
C01347=1063.081,72.830,427.215,172.149,28.417,155.243
C01348=1063.074,72.580,427.233,172.147,28.414,155.243
C01349=1063.069,72.331,427.251,172.147,28.412,155.242
C01350=1063.063,72.081,427.269,172.145,28.409,155.242
C01351=1063.057,71.832,427.286,172.144,28.406,155.242
C01352=1063.050,71.583,427.304,172.142,28.404,155.241
C01353=1063.045,71.334,427.321,172.140,28.401,155.241
C01354=1063.039,71.084,427.339,172.139,28.398,155.241
C01355=1063.033,70.835,427.357,172.137,28.395,155.240
C01356=1063.027,70.585,427.375,172.137,28.393,155.240
C01357=1063.021,70.337,427.392,172.135,28.390,155.239
C01358=1063.015,70.088,427.409,172.133,28.387,155.239
C01359=1063.009,69.838,427.427,172.132,28.385,155.239
C01360=1063.004,69.589,427.445,172.130,28.382,155.238
C01361=1062.998,69.339,427.463,172.129,28.380,155.238
C01362=1062.991,69.090,427.479,172.127,28.377,155.238
C01363=1062.985,68.841,427.497,172.126,28.374,155.237
C01364=1062.980,68.592,427.515,172.125,28.371,155.237
C01365=1062.973,68.342,427.532,172.123,28.369,155.236
C01366=1062.967,68.093,427.550,172.122,28.366,155.236
C01367=1062.962,67.843,427.567,172.120,28.364,155.236
C01368=1062.955,67.594,427.584,172.118,28.361,155.235
C01369=1062.950,67.345,427.602,172.117,28.358,155.235
C01370=1062.944,67.095,427.620,172.116,28.356,155.234
C01371=1062.937,66.847,427.637,172.115,28.353,155.234
C01372=1062.931,66.597,427.654,172.113,28.351,155.234
C01373=1062.926,66.348,427.672,172.111,28.348,155.233
C01374=1062.920,66.098,427.688,172.110,28.345,155.233
C01375=1062.914,65.849,427.706,172.108,28.342,155.233
C01376=1062.908,65.600,427.724,172.107,28.339,155.232
C01377=1062.901,65.350,427.741,172.106,28.337,155.232
C01378=1062.896,65.101,427.759,172.104,28.335,155.231
C01379=1062.890,64.852,427.775,172.103,28.332,155.231
C01380=1062.884,64.602,427.793,172.101,28.329,155.231
C01381=1062.878,64.353,427.810,172.100,28.326,155.230
C01382=1062.871,64.104,427.828,172.098,28.323,155.230
C01383=1062.866,63.854,427.845,172.096,28.321,155.230
C01384=1062.860,63.605,427.862,172.096,28.319,155.229
C01385=1062.853,63.356,427.879,172.094,28.316,155.229
C01386=1062.848,63.107,427.897,172.093,28.313,155.228
C01387=1062.841,62.857,427.913,172.091,28.311,155.228
C01388=1062.834,62.573,427.932,172.089,28.308,155.228
C01389=1062.827,62.289,427.953,172.088,28.305,155.227
C01390=1062.821,62.005,427.972,172.086,28.302,155.227
C01391=1062.813,61.721,427.992,172.085,28.299,155.226
C01392=1062.807,61.471,428.008,172.083,28.296,155.226
C01393=1062.801,61.222,428.026,172.082,28.294,155.226
C01394=1062.795,60.973,428.043,172.080,28.291,155.225
C01395=1062.788,60.723,428.060,172.078,28.289,155.225
C01396=1062.783,60.474,428.077,172.077,28.286,155.224
C01397=1062.777,60.225,428.094,172.075,28.283,155.224
C01398=1062.771,59.975,428.111,172.074,28.281,155.224
C01399=1062.765,59.726,428.128,172.073,28.278,155.223
C01400=1062.759,59.477,428.145,172.071,28.275,155.223
C01401=1062.752,59.227,428.163,172.070,28.273,155.223
C01402=1062.746,58.978,428.180,172.068,28.270,155.222
C01403=1062.740,58.729,428.196,172.067,28.268,155.222
C01404=1062.734,58.479,428.214,172.066,28.265,155.221
C01405=1062.728,58.230,428.230,172.064,28.262,155.221
C01406=1062.722,57.981,428.247,172.063,28.260,155.221
C01407=1062.716,57.731,428.264,172.061,28.257,155.220
C01408=1062.710,57.482,428.281,172.060,28.255,155.220
C01409=1062.705,57.232,428.298,172.058,28.252,155.220
C01410=1062.698,56.983,428.315,172.056,28.250,155.219
C01411=1062.692,56.734,428.332,172.056,28.247,155.219
C01412=1062.686,56.484,428.349,172.054,28.244,155.219
C01413=1062.679,56.235,428.366,172.053,28.241,155.218
C01414=1062.673,55.986,428.383,172.051,28.239,155.218
C01415=1062.668,55.737,428.400,172.049,28.236,155.217
C01416=1062.662,55.487,428.417,172.048,28.234,155.217
C01417=1062.655,55.237,428.433,172.046,28.231,155.217
C01418=1062.650,54.988,428.451,172.045,28.229,155.216
C01419=1062.644,54.739,428.467,172.044,28.226,155.216
C01420=1062.637,54.489,428.484,172.042,28.223,155.216
C01421=1062.632,54.240,428.501,172.041,28.220,155.215
C01422=1062.626,53.991,428.518,172.039,28.218,155.215
C01423=1062.620,53.742,428.534,172.038,28.215,155.215
C01424=1062.613,53.492,428.552,172.037,28.213,155.214
C01425=1062.608,53.243,428.569,172.035,28.210,155.214
C01426=1062.602,52.993,428.585,172.034,28.207,155.213
C01427=1062.595,52.744,428.602,172.032,28.205,155.213
C01428=1062.590,52.495,428.619,172.031,28.202,155.213
C01429=1062.583,52.245,428.636,172.029,28.199,155.212
C01430=1062.577,51.996,428.652,172.027,28.197,155.212
C01431=1062.572,51.746,428.669,172.027,28.194,155.211
C01432=1062.566,51.498,428.686,172.025,28.192,155.211
C01433=1062.559,51.248,428.703,172.024,28.189,155.211
C01434=1062.553,50.998,428.719,172.022,28.186,155.210
C01435=1062.548,50.749,428.737,172.021,28.183,155.210
C01436=1062.542,50.500,428.753,172.019,28.181,155.210
C01437=1062.536,50.250,428.769,172.018,28.179,155.209
C01438=1062.531,50.001,428.787,172.017,28.176,155.209
C01439=1062.524,49.751,428.803,172.015,28.173,155.208
C01440=1062.518,49.502,428.820,172.014,28.170,155.208
C01441=1062.512,49.253,428.836,172.012,28.167,155.208
C01442=1062.507,49.004,428.853,172.010,28.165,155.207
C01443=1062.501,48.754,428.870,172.010,28.163,155.207
C01444=1062.495,48.505,428.886,172.008,28.160,155.207
C01445=1062.488,48.255,428.902,172.007,28.157,155.206
C01446=1062.483,48.006,428.920,172.005,28.154,155.206
C01447=1062.477,47.757,428.936,172.003,28.152,155.205
C01448=1062.471,47.507,428.953,172.002,28.149,155.205
C01449=1062.465,47.258,428.969,172.000,28.146,155.205
C01450=1062.459,47.009,428.986,172.000,28.144,155.204
C01451=1062.453,46.759,429.003,171.998,28.141,155.204
C01452=1062.446,46.475,429.022,171.997,28.138,155.203
C01453=1062.440,46.190,429.040,171.995,28.135,155.203
C01454=1062.433,45.906,429.059,171.993,28.132,155.203
C01455=1062.426,45.621,429.078,171.991,28.129,155.202
C01456=1062.420,45.373,429.095,171.990,28.126,155.202
C01457=1062.415,45.123,429.112,171.989,28.124,155.201
C01458=1062.409,44.874,429.128,171.987,28.121,155.201
C01459=1062.403,44.624,429.144,171.986,28.119,155.201
C01460=1062.397,44.375,429.160,171.984,28.116,155.200
C01461=1062.391,44.125,429.177,171.982,28.113,155.200
C01462=1062.386,43.876,429.194,171.982,28.110,155.200
C01463=1062.379,43.627,429.211,171.980,28.108,155.199
C01464=1062.373,43.377,429.227,171.979,28.105,155.199
C01465=1062.367,43.128,429.243,171.977,28.103,155.198
C01466=1062.361,42.878,429.260,171.976,28.100,155.198
C01467=1062.355,42.629,429.276,171.974,28.098,155.198
C01468=1062.349,42.380,429.292,171.972,28.095,155.197
C01469=1062.343,42.130,429.308,171.972,28.092,155.197
C01470=1062.337,41.881,429.325,171.970,28.089,155.197
C01471=1062.331,41.632,429.341,171.969,28.087,155.196
C01472=1062.325,41.382,429.357,171.967,28.084,155.196
C01473=1062.319,41.133,429.373,171.965,28.082,155.196
C01474=1062.313,40.884,429.390,171.964,28.079,155.195
C01475=1062.307,40.633,429.406,171.963,28.077,155.195
C01476=1062.301,40.384,429.423,171.962,28.074,155.194
C01477=1062.295,40.135,429.439,171.960,28.071,155.194
C01478=1062.289,39.885,429.455,171.958,28.069,155.194
C01479=1062.283,39.636,429.471,171.957,28.066,155.193
C01480=1062.277,39.387,429.488,171.955,28.063,155.193
C01481=1062.271,39.137,429.504,171.954,28.061,155.193
C01482=1062.265,38.888,429.520,171.953,28.059,155.192
C01483=1062.259,38.639,429.536,171.952,28.056,155.192
C01484=1062.253,38.389,429.553,171.950,28.053,155.191
C01485=1062.247,38.140,429.569,171.948,28.051,155.191
C01486=1062.241,37.891,429.585,171.947,28.048,155.191
C01487=1062.236,37.641,429.601,171.945,28.045,155.190
C01488=1062.230,37.391,429.617,171.945,28.043,155.190
C01489=1062.223,37.142,429.633,171.943,28.040,155.190
C01490=1062.217,36.893,429.649,171.941,28.037,155.189
C01491=1062.211,36.644,429.665,171.940,28.035,155.189
C01492=1062.205,36.394,429.681,171.938,28.032,155.189
C01493=1062.199,36.145,429.698,171.937,28.030,155.188
C01494=1062.193,35.895,429.713,171.935,28.027,155.188
C01495=1062.186,35.645,429.729,171.934,28.025,155.188
C01496=1062.180,35.396,429.745,171.933,28.023,155.187
C01497=1062.174,35.147,429.762,171.931,28.020,155.187
C01498=1062.168,34.897,429.778,171.930,28.017,155.186
C01499=1062.162,34.648,429.794,171.928,28.015,155.186
C01500=1062.156,34.398,429.809,171.927,28.012,155.186
C01501=1062.150,34.149,429.825,171.925,28.010,155.186
C01502=1062.144,33.899,429.842,171.924,28.007,155.185
C01503=1062.137,33.650,429.857,171.923,28.004,155.185
C01504=1062.132,33.400,429.873,171.921,28.002,155.184
C01505=1062.126,33.151,429.889,171.920,27.999,155.184
C01506=1062.120,32.902,429.905,171.918,27.996,155.184
C01507=1062.114,32.652,429.922,171.916,27.994,155.183
C01508=1062.108,32.403,429.937,171.915,27.991,155.183
C01509=1062.102,32.153,429.953,171.914,27.989,155.183
C01510=1062.096,31.905,429.969,171.913,27.987,155.182
C01511=1062.090,31.655,429.985,171.911,27.984,155.182
C01512=1062.084,31.406,430.000,171.909,27.982,155.182
C01513=1062.078,31.156,430.016,171.908,27.979,155.181
C01514=1062.072,30.907,430.032,171.906,27.976,155.181
C01515=1062.066,30.657,430.048,171.905,27.974,155.181
C01516=1062.059,30.373,430.066,171.903,27.971,155.180
C01517=1062.052,30.089,430.084,171.902,27.967,155.180
C01518=1062.045,29.804,430.102,171.900,27.965,155.179
C01519=1062.038,29.520,430.120,171.899,27.962,155.179
C01520=1062.032,29.270,430.136,171.897,27.960,155.179
C01521=1062.026,29.021,430.152,171.895,27.957,155.178
C01522=1062.020,28.771,430.168,171.894,27.954,155.178
C01523=1062.014,28.522,430.183,171.893,27.952,155.178
C01524=1062.009,28.273,430.199,171.892,27.949,155.177
C01525=1062.002,28.023,430.214,171.890,27.947,155.177
C01526=1061.996,27.774,430.230,171.888,27.944,155.176
C01527=1061.991,27.524,430.246,171.887,27.941,155.176
C01528=1061.984,27.275,430.262,171.885,27.939,155.176
C01529=1061.978,27.026,430.278,171.884,27.936,155.175
C01530=1061.972,26.776,430.293,171.883,27.934,155.175
C01531=1061.966,26.527,430.309,171.882,27.931,155.175
C01532=1061.960,26.277,430.325,171.880,27.929,155.174
C01533=1061.953,26.028,430.340,171.878,27.926,155.174
C01534=1061.948,25.778,430.356,171.877,27.924,155.174
C01535=1061.942,25.529,430.371,171.875,27.921,155.173
C01536=1061.936,25.279,430.387,171.874,27.918,155.173
C01537=1061.929,25.030,430.402,171.873,27.916,155.173
C01538=1061.924,24.780,430.418,171.871,27.914,155.172
C01539=1061.917,24.531,430.434,171.870,27.911,155.172
C01540=1061.911,24.281,430.449,171.868,27.909,155.172
C01541=1061.905,24.032,430.465,171.867,27.906,155.171
C01542=1061.899,23.782,430.480,171.865,27.904,155.171
C01543=1061.892,23.533,430.496,171.863,27.901,155.171
C01544=1061.887,23.284,430.511,171.863,27.899,155.170
C01545=1061.881,23.034,430.526,171.861,27.896,155.170
C01546=1061.875,22.785,430.542,171.860,27.894,155.170
C01547=1061.868,22.535,430.557,171.858,27.891,155.169
C01548=1061.862,22.286,430.574,171.857,27.889,155.169
C01549=1061.856,22.036,430.589,171.855,27.886,155.169
C01550=1061.851,21.787,430.604,171.853,27.884,155.168
C01551=1061.844,21.538,430.619,171.852,27.881,155.168
C01552=1061.839,21.288,430.635,171.851,27.879,155.168
C01553=1061.832,21.039,430.651,171.850,27.876,155.167
C01554=1061.826,20.789,430.666,171.848,27.874,155.167
C01555=1061.820,20.539,430.681,171.846,27.871,155.167
C01556=1061.815,20.291,430.697,171.845,27.869,155.166
C01557=1061.808,20.041,430.712,171.843,27.866,155.166
C01558=1061.803,19.791,430.727,171.842,27.864,155.166
C01559=1061.796,19.542,430.743,171.841,27.861,155.165
C01560=1061.790,19.292,430.758,171.839,27.859,155.165
C01561=1061.784,19.043,430.773,171.838,27.856,155.165
C01562=1061.778,18.794,430.789,171.836,27.854,155.164
C01563=1061.771,18.544,430.804,171.835,27.851,155.164
C01564=1061.766,18.294,430.819,171.833,27.849,155.164
C01565=1061.759,18.045,430.834,171.832,27.846,155.163
C01566=1061.754,17.796,430.850,171.830,27.843,155.163
C01567=1061.748,17.547,430.865,171.829,27.841,155.162
C01568=1061.741,17.297,430.880,171.828,27.839,155.162
C01569=1061.736,17.047,430.896,171.826,27.836,155.162
C01570=1061.729,16.798,430.911,171.825,27.834,155.162
C01571=1061.723,16.549,430.926,171.823,27.831,155.161
C01572=1061.718,16.299,430.941,171.821,27.829,155.161
C01573=1061.711,16.049,430.956,171.820,27.826,155.161
C01574=1061.705,15.800,430.971,171.818,27.823,155.160
C01575=1061.699,15.551,430.987,171.818,27.821,155.160
C01576=1061.693,15.301,431.002,171.816,27.819,155.160
C01577=1061.687,15.052,431.017,171.814,27.816,155.159
C01578=1061.681,14.802,431.033,171.813,27.814,155.159
C01579=1061.675,14.553,431.047,171.811,27.811,155.159
C01580=1061.668,14.270,431.064,171.810,27.808,155.158
C01581=1061.661,13.987,431.082,171.808,27.806,155.158
C01582=1061.654,13.704,431.099,171.807,27.803,155.157
C01583=1061.647,13.420,431.115,171.805,27.800,155.157
C01584=1061.641,13.171,431.132,171.804,27.798,155.157
C01585=1061.634,12.921,431.147,171.802,27.795,155.157
C01586=1061.629,12.672,431.161,171.800,27.793,155.156
C01587=1061.622,12.423,431.176,171.799,27.790,155.156
C01588=1061.616,12.173,431.191,171.797,27.788,155.156
C01589=1061.609,11.923,431.206,171.796,27.785,155.155
C01590=1061.604,11.675,431.221,171.794,27.783,155.155
C01591=1061.597,11.425,431.235,171.793,27.781,155.155
C01592=1061.592,11.175,431.251,171.792,27.778,155.154
C01593=1061.585,10.925,431.266,171.790,27.776,155.154
C01594=1061.579,10.676,431.281,171.789,27.774,155.154
C01595=1061.573,10.427,431.295,171.787,27.771,155.153
C01596=1061.567,10.177,431.310,171.785,27.769,155.153
C01597=1061.561,9.928,431.325,171.784,27.766,155.153
C01598=1061.555,9.678,431.340,171.782,27.764,155.152
C01599=1061.548,9.429,431.355,171.781,27.761,155.152
C01600=1061.542,9.179,431.370,171.780,27.759,155.152
C01601=1061.536,8.930,431.384,171.778,27.756,155.151
C01602=1061.530,8.680,431.399,171.777,27.754,155.151
C01603=1061.524,8.430,431.415,171.775,27.752,155.151
C01604=1061.518,8.182,431.429,171.774,27.749,155.150
C01605=1061.512,7.932,431.444,171.772,27.747,155.150
C01606=1061.505,7.682,431.459,171.770,27.745,155.150
C01607=1061.500,7.433,431.474,171.769,27.742,155.150
C01608=1061.493,7.184,431.489,171.767,27.740,155.149
C01609=1061.487,6.934,431.504,171.767,27.738,155.149
C01610=1061.481,6.685,431.518,171.765,27.735,155.149
C01611=1061.475,6.435,431.533,171.764,27.732,155.148
C01612=1061.469,6.185,431.548,171.762,27.730,155.148
C01613=1061.463,5.936,431.562,171.760,27.727,155.148
C01614=1061.456,5.686,431.577,171.759,27.725,155.147
C01615=1061.451,5.437,431.592,171.757,27.723,155.147
C01616=1061.444,5.188,431.607,171.756,27.720,155.147
C01617=1061.438,4.938,431.622,171.754,27.718,155.146
C01618=1061.433,4.689,431.637,171.753,27.716,155.146
C01619=1061.427,4.439,431.651,171.752,27.713,155.146
C01620=1061.420,4.189,431.666,171.750,27.711,155.145
C01621=1061.415,3.940,431.681,171.749,27.708,155.145
C01622=1061.408,3.690,431.695,171.747,27.706,155.145
C01623=1061.402,3.441,431.710,171.745,27.703,155.145
C01624=1061.396,3.191,431.724,171.744,27.701,155.144
C01625=1061.391,2.942,431.739,171.742,27.698,155.144
C01626=1061.384,2.692,431.754,171.741,27.696,155.144
C01627=1061.378,2.443,431.769,171.739,27.694,155.143
C01628=1061.372,2.194,431.783,171.738,27.691,155.143
C01629=1061.366,1.944,431.798,171.737,27.689,155.143
C01630=1061.360,1.695,431.812,171.735,27.687,155.142
C01631=1061.354,1.445,431.827,171.734,27.684,155.142
C01632=1061.348,1.196,431.842,171.732,27.682,155.142
C01633=1061.342,0.946,431.856,171.731,27.679,155.141
C01634=1061.336,0.697,431.871,171.729,27.676,155.141
C01635=1061.330,0.447,431.885,171.727,27.674,155.141
C01636=1061.324,0.197,431.900,171.726,27.672,155.141
C01637=1061.318,-0.052,431.914,171.724,27.670,155.140
C01638=1061.312,-0.302,431.929,171.724,27.667,155.140
C01639=1061.306,-0.551,431.943,171.722,27.665,155.140
C01640=1061.300,-0.801,431.958,171.720,27.663,155.139
C01641=1061.294,-1.050,431.973,171.719,27.660,155.139
C01642=1061.288,-1.300,431.987,171.717,27.657,155.139
C01643=1061.282,-1.549,432.001,171.716,27.655,155.138
C01644=1061.275,-1.830,432.018,171.714,27.652,155.138
C01645=1061.269,-2.111,432.034,171.713,27.650,155.138
C01646=1061.262,-2.392,432.050,171.711,27.647,155.137
C01647=1061.255,-2.673,432.067,171.709,27.644,155.137
C01648=1061.249,-2.923,432.081,171.708,27.642,155.137
C01649=1061.243,-3.172,432.096,171.706,27.639,155.136
C01650=1061.237,-3.422,432.110,171.705,27.637,155.136
C01651=1061.231,-3.671,432.124,171.703,27.635,155.136
C01652=1061.225,-3.921,432.138,171.702,27.633,155.135
C01653=1061.219,-4.170,432.153,171.700,27.630,155.135
C01654=1061.212,-4.420,432.167,171.698,27.627,155.135
C01655=1061.206,-4.670,432.181,171.697,27.625,155.135
C01656=1061.200,-4.919,432.196,171.695,27.623,155.134
C01657=1061.194,-5.169,432.210,171.694,27.621,155.134
C01658=1061.187,-5.418,432.224,171.692,27.618,155.134
C01659=1061.181,-5.668,432.238,171.691,27.616,155.133
C01660=1061.175,-5.917,432.253,171.690,27.614,155.133
C01661=1061.169,-6.167,432.267,171.688,27.612,155.133
C01662=1061.163,-6.416,432.281,171.687,27.609,155.133
C01663=1061.157,-6.666,432.295,171.685,27.607,155.132
C01664=1061.150,-6.915,432.309,171.683,27.604,155.132
C01665=1061.144,-7.165,432.324,171.682,27.602,155.132
C01666=1061.139,-7.415,432.338,171.680,27.600,155.131
C01667=1061.133,-7.664,432.352,171.679,27.598,155.131
C01668=1061.126,-7.914,432.366,171.677,27.595,155.131
C01669=1061.120,-8.163,432.380,171.675,27.593,155.131
C01670=1061.114,-8.413,432.395,171.674,27.590,155.130
C01671=1061.108,-8.662,432.409,171.672,27.588,155.130
C01672=1061.102,-8.912,432.423,171.672,27.586,155.130
C01673=1061.096,-9.161,432.437,171.670,27.584,155.129
C01674=1061.089,-9.411,432.451,171.668,27.582,155.129
C01675=1061.084,-9.660,432.465,171.667,27.579,155.129
C01676=1061.078,-9.909,432.479,171.665,27.577,155.129
C01677=1061.071,-10.159,432.493,171.663,27.575,155.128
C01678=1061.065,-10.409,432.507,171.662,27.572,155.128
C01679=1061.058,-10.658,432.521,171.660,27.570,155.128
C01680=1061.053,-10.908,432.535,171.659,27.567,155.127
C01681=1061.047,-11.157,432.549,171.657,27.565,155.127
C01682=1061.040,-11.407,432.563,171.656,27.563,155.127
C01683=1061.035,-11.656,432.577,171.654,27.561,155.127
C01684=1061.029,-11.907,432.591,171.652,27.558,155.126
C01685=1061.022,-12.155,432.605,171.651,27.556,155.126
C01686=1061.017,-12.405,432.619,171.650,27.554,155.126
C01687=1061.011,-12.655,432.634,171.648,27.552,155.125
C01688=1061.004,-12.904,432.648,171.647,27.549,155.125
C01689=1060.999,-13.153,432.661,171.645,27.547,155.125
C01690=1060.992,-13.403,432.675,171.644,27.545,155.125
C01691=1060.986,-13.653,432.689,171.642,27.542,155.124
C01692=1060.980,-13.902,432.704,171.641,27.540,155.124
C01693=1060.974,-14.152,432.717,171.639,27.538,155.124
C01694=1060.968,-14.401,432.731,171.637,27.535,155.124
C01695=1060.962,-14.652,432.745,171.636,27.533,155.123
C01696=1060.956,-14.900,432.759,171.634,27.531,155.123
C01697=1060.950,-15.150,432.773,171.633,27.529,155.123
C01698=1060.943,-15.400,432.787,171.631,27.526,155.122
C01699=1060.938,-15.649,432.801,171.629,27.524,155.122
C01700=1060.932,-15.899,432.814,171.628,27.522,155.122
C01701=1060.925,-16.149,432.827,171.626,27.519,155.122
C01702=1060.919,-16.398,432.842,171.625,27.517,155.121
C01703=1060.913,-16.647,432.855,171.624,27.515,155.121
C01704=1060.907,-16.897,432.870,171.622,27.513,155.121
C01705=1060.901,-17.146,432.883,171.621,27.511,155.121
C01706=1060.894,-17.396,432.896,171.619,27.509,155.120
C01707=1060.888,-17.646,432.910,171.617,27.507,155.120
C01708=1060.881,-17.925,432.926,171.616,27.504,155.120
C01709=1060.874,-18.204,432.941,171.613,27.501,155.120
C01710=1060.868,-18.484,432.956,171.612,27.499,155.119
C01711=1060.860,-18.764,432.972,171.610,27.497,155.119
C01712=1060.854,-19.013,432.985,171.609,27.494,155.119
C01713=1060.849,-19.263,432.999,171.607,27.492,155.118
C01714=1060.842,-19.513,433.013,171.605,27.490,155.118
C01715=1060.837,-19.762,433.026,171.604,27.488,155.118
C01716=1060.830,-20.012,433.040,171.602,27.485,155.118
C01717=1060.824,-20.260,433.054,171.601,27.483,155.117
C01718=1060.818,-20.510,433.068,171.599,27.481,155.117
C01719=1060.811,-20.760,433.081,171.597,27.479,155.117
C01720=1060.805,-21.009,433.094,171.597,27.477,155.117
C01721=1060.799,-21.259,433.109,171.595,27.474,155.116
C01722=1060.793,-21.509,433.122,171.593,27.473,155.116
C01723=1060.788,-21.758,433.136,171.592,27.470,155.116
C01724=1060.781,-22.007,433.149,171.590,27.468,155.116
C01725=1060.774,-22.257,433.163,171.589,27.466,155.115
C01726=1060.769,-22.507,433.177,171.587,27.464,155.115
C01727=1060.763,-22.756,433.190,171.585,27.461,155.115
C01728=1060.757,-23.006,433.202,171.584,27.459,155.115
C01729=1060.751,-23.256,433.216,171.582,27.457,155.114
C01730=1060.745,-23.506,433.230,171.581,27.454,155.114
C01731=1060.738,-23.755,433.243,171.579,27.453,155.114
C01732=1060.733,-24.004,433.257,171.577,27.450,155.114
C01733=1060.727,-24.254,433.270,171.576,27.448,155.113
C01734=1060.720,-24.504,433.284,171.574,27.446,155.113
C01735=1060.714,-24.753,433.298,171.573,27.444,155.113
C01736=1060.708,-25.003,433.311,171.571,27.441,155.113
C01737=1060.702,-25.252,433.324,171.569,27.439,155.112
C01738=1060.696,-25.501,433.338,171.568,27.437,155.112
C01739=1060.690,-25.751,433.351,171.566,27.435,155.112
C01740=1060.684,-26.001,433.364,171.564,27.433,155.112
C01741=1060.678,-26.251,433.378,171.563,27.431,155.111
C01742=1060.672,-26.500,433.392,171.561,27.428,155.111
C01743=1060.666,-26.749,433.405,171.560,27.426,155.111
C01744=1060.660,-26.999,433.418,171.559,27.424,155.110
C01745=1060.653,-27.249,433.432,171.557,27.422,155.110
C01746=1060.648,-27.499,433.445,171.556,27.420,155.110
C01747=1060.641,-27.748,433.458,171.554,27.418,155.110
C01748=1060.635,-27.997,433.471,171.552,27.416,155.110
C01749=1060.629,-28.247,433.485,171.551,27.414,155.109
C01750=1060.622,-28.496,433.498,171.549,27.412,155.109
C01751=1060.616,-28.746,433.511,171.548,27.409,155.109
C01752=1060.610,-28.996,433.524,171.546,27.408,155.109
C01753=1060.604,-29.245,433.537,171.544,27.405,155.108
C01754=1060.598,-29.494,433.551,171.543,27.403,155.108
C01755=1060.592,-29.745,433.564,171.541,27.401,155.108
C01756=1060.586,-29.994,433.577,171.539,27.399,155.108
C01757=1060.579,-30.244,433.591,171.538,27.397,155.107
C01758=1060.574,-30.493,433.603,171.536,27.395,155.107
C01759=1060.567,-30.743,433.617,171.535,27.393,155.107
C01760=1060.561,-30.992,433.630,171.533,27.391,155.107
C01761=1060.555,-31.241,433.643,171.531,27.388,155.107
C01762=1060.548,-31.492,433.656,171.530,27.387,155.106
C01763=1060.542,-31.741,433.669,171.528,27.384,155.106
C01764=1060.536,-31.990,433.683,171.527,27.382,155.106
C01765=1060.530,-32.240,433.695,171.525,27.380,155.106
C01766=1060.524,-32.490,433.708,171.523,27.378,155.105
C01767=1060.518,-32.739,433.722,171.522,27.376,155.105
C01768=1060.512,-32.989,433.735,171.520,27.374,155.105
C01769=1060.506,-33.238,433.748,171.518,27.372,155.105
C01770=1060.500,-33.489,433.761,171.517,27.369,155.104
C01771=1060.494,-33.738,433.774,171.515,27.368,155.104
C01772=1060.487,-34.016,433.788,171.514,27.366,155.104
C01773=1060.480,-34.295,433.803,171.512,27.363,155.104
C01774=1060.473,-34.574,433.818,171.509,27.361,155.104
C01775=1060.466,-34.852,433.832,171.508,27.358,155.103
C01776=1060.460,-35.102,433.845,171.506,27.356,155.103
C01777=1060.454,-35.351,433.858,171.505,27.354,155.103
C01778=1060.448,-35.601,433.871,171.503,27.352,155.103
C01779=1060.442,-35.851,433.884,171.501,27.350,155.102
C01780=1060.436,-36.101,433.897,171.500,27.348,155.102
C01781=1060.429,-36.350,433.910,171.498,27.346,155.102
C01782=1060.424,-36.600,433.922,171.496,27.344,155.102
C01783=1060.417,-36.849,433.936,171.495,27.342,155.102
C01784=1060.412,-37.099,433.949,171.493,27.340,155.101
C01785=1060.406,-37.348,433.962,171.491,27.338,155.101
C01786=1060.400,-37.598,433.975,171.490,27.336,155.101
C01787=1060.394,-37.848,433.988,171.488,27.333,155.101
C01788=1060.388,-38.097,434.001,171.487,27.332,155.100
C01789=1060.382,-38.347,434.014,171.485,27.329,155.100
C01790=1060.376,-38.597,434.026,171.483,27.328,155.100
C01791=1060.369,-38.846,434.039,171.482,27.325,155.100
C01792=1060.363,-39.095,434.052,171.480,27.324,155.100
C01793=1060.356,-39.345,434.065,171.478,27.321,155.099
C01794=1060.350,-39.595,434.078,171.477,27.320,155.099
C01795=1060.344,-39.845,434.090,171.475,27.317,155.099
C01796=1060.338,-40.094,434.104,171.474,27.316,155.099
C01797=1060.331,-40.344,434.116,171.472,27.313,155.099
C01798=1060.325,-40.593,434.129,171.470,27.312,155.098
C01799=1060.319,-40.843,434.141,171.469,27.309,155.098
C01800=1060.313,-41.093,434.154,171.467,27.308,155.098
C01801=1060.307,-41.342,434.167,171.465,27.306,155.098
C01802=1060.301,-41.592,434.179,171.464,27.304,155.098
C01803=1060.295,-41.842,434.192,171.462,27.302,155.097
C01804=1060.288,-42.091,434.205,171.460,27.300,155.097
C01805=1060.283,-42.341,434.218,171.459,27.298,155.097
C01806=1060.276,-42.590,434.230,171.457,27.296,155.097
C01807=1060.270,-42.840,434.243,171.455,27.294,155.097
C01808=1060.264,-43.090,434.255,171.454,27.292,155.096
C01809=1060.258,-43.339,434.268,171.452,27.290,155.096
C01810=1060.252,-43.589,434.281,171.451,27.288,155.096
C01811=1060.245,-43.838,434.293,171.449,27.286,155.096
C01812=1060.239,-44.088,434.306,171.447,27.284,155.096
C01813=1060.233,-44.337,434.319,171.446,27.282,155.095
C01814=1060.228,-44.587,434.331,171.444,27.280,155.095
C01815=1060.221,-44.836,434.343,171.442,27.279,155.095
C01816=1060.215,-45.086,434.356,171.441,27.277,155.095
C01817=1060.209,-45.335,434.369,171.439,27.275,155.095
C01818=1060.203,-45.585,434.381,171.437,27.273,155.094
